ACTION OpenSeperator_action:
ST03_557_Y70_1.MoveInit:=TRUE;		(* Zuführung Vereinzler AST/GST *)
END_ACTION

ACTION Kamera_nicht_bb_entry:
MessageHandler.ClearMessageLines(sVisu:=Visu.Message);
END_ACTION

ACTION Kamera_nicht_bb_action:
MessageHandler.Msg.ID:='PM152';
MessageHandler.Msg.Name:='Check Camera';
MessageHandler.Msg.Text:='Sesopart Kamera ist nicht betriebsbereit';
MessageHandler.Msg.Color:=Color.red;
MessageHandler.Msg.Station:=1;


MessageHandler(
	Prio:=2, 							(*1=highest, .. , 4=lowest*)
	Btn1Addr:=ADR(MsgOk),			(*Address of Button1 , if Zero then Button is unvisible*)
	Btn2Addr:=,						(*Address of Button2 , if Zero then Button is unvisible*)
	sVisu:=Visu.Message);
END_ACTION

ACTION Kamera_nicht_bb_exit:
MsgOk:=FALSE;
MsgCancel:=FALSE;
ST02_DT_95_A1.b_quitt:=TRUE;
END_ACTION

ACTION Wait_for_Part_entry:
ProcessMessage01:='';
Delay.IN:=FALSE;
Delay();
END_ACTION

ACTION Wait_for_Part_action:
ProcessMessage01:='1IM9';(*warte auf Teil in Stopper*)
Delay.IN:=ST03_556_B69_6.BitInToCheck; 		(*  ISK an Stopper.*)
Delay.PT:=T#500ms;
Delay();
END_ACTION

ACTION Wait_for_Part_exit:
ProcessMessage01:='';
END_ACTION

ACTION Close_Seperator_action:
ST03_557_Y70_1.MoveWork:=TRUE;		(*Zuführung Vereinzler AST/GST *)
END_ACTION

ACTION Open_Stopper_action:
ST03_557_Y70_2.MoveWork:=TRUE;		(* Züführung Stopper AST/GST *)
END_ACTION

ACTION Wait_for_Part__entry:
ProcessMessage01:='';
Delay(IN:=FALSE);
END_ACTION

ACTION Wait_for_Part__action:
ProcessMessage01:='1IM10';(*warte auf Teil in Abholposition*)
Delay(	IN:=	ST03_Init_AbholPos.RoboPos31,
		PT:=T#500ms);
END_ACTION

ACTION Wait_for_Part__exit:
ProcessMessage01:='';
Delay(IN:=FALSE);
END_ACTION

ACTION Close_Stopper_action:
ST03_557_Y70_2.MoveInit:=TRUE;		(* Züführung Stopper AST/GST *)
END_ACTION

ACTION Open_Seperator_action:
ST03_557_Y70_1.MoveInit:=TRUE;		(* Zuführung Vereinzler AST/GST *)
END_ACTION

ACTION Robot01_Pos31_action:
Robot01.PosNo:=POS_WT_POS1;
Robot01.PosOffset:=gRobotOffset;
Robot01.Override:=MP.ST00.Override;
Robot01.SetToolOn:=FALSE;
Robot01.SetToolOff:=TRUE;
Robot01.ExecuteMove:=TRUE;
END_ACTION

ACTION Robot01_Pos31_exit:
gRob01GripState:=PART_CAM;
FOR i:=1 TO NO_OF_RESULT BY 1 DO
	Result[i]:=0;
END_FOR
END_ACTION

ACTION Robot01_Pos41_entry:
RepeatCounter:=0;
END_ACTION

ACTION Robot01_Pos41_action:
Robot01.PosNo:=POS_CAM_POS1;
Robot01.PosOffset:=gRobotOffset;
Robot01.Override:=MP.ST00.Override;
Robot01.SetToolOn:=FALSE;
Robot01.SetToolOff:=TRUE;
Robot01.ExecuteMove:=TRUE;
Pos:=1;
END_ACTION

ACTION Robot01_Pos45_entry:
RepeatCounter:=0;
END_ACTION

ACTION Robot01_Pos45_action:
Robot01.PosNo:=POS_CAM_POS2;
Robot01.PosOffset:=gRobotOffset;
Robot01.Override:=MP.ST00.Override;
Robot01.SetToolOn:=FALSE;
Robot01.SetToolOff:=TRUE;
Robot01.ExecuteMove:=TRUE;
Pos:=2;
END_ACTION

ACTION Start_Sensopart_action:
ST03_8_100_A1.JobNo := TD.Sensopart_CamProgNo ;
ST03_8_100_A1.st_ctrl_in.b_start := TRUE;
END_ACTION

ACTION WaitDone_entry:
ST03_8_100_A1.st_ctrl_in.b_start := FALSE;
RepeatCounter:=RepeatCounter+1;
END_ACTION

ACTION ResultCam_entry:
IF 	(ST03_8_100_A1.b_Kam_Pruef_IO AND	 (*Kamera Farberkennung*)
	NOT ST03_8_100_A1.b_Kam_Pruef_NIO) THEN
	Result[Pos]:=RESULT_OK;
ELSE
	Result[Pos]:=RESULT_NOK;
END_IF
END_ACTION

ACTION Result2_entry:
FOR i:=1 TO NO_OF_RESULT BY 1 DO
	Result[i]:=RESULT_OK;
END_FOR
END_ACTION

ACTION Result_Counter_entry:
FOR i:=100 TO 2 BY-1 DO
   	NokPercent[i] := NokPercent[i-1];
END_FOR

ResultOk:=TRUE;
FOR i:=1 TO NO_OF_RESULT BY 1 DO
	IF	ResultOk AND Result[i] = RESULT_NOK 	THEN
		ResultOk:=FALSE;
	END_IF
END_FOR

IF 	ResultOk OR
	CamAlwaysOK THEN		(*schreibt immer NOK nur zum Testen*)
	NokCounter:=0;
	NokPercent[1] := FALSE;
	gRob01GripState:=PART_OK;
ELSE
	NokCounter:=NokCounter+1;
	NokPercent[1] := TRUE;
	gRob01GripState:=PART_NOK;
END_IF
END_ACTION

ACTION Msg_Cam_entry:
MessageHandler.ClearMessageLines(sVisu:=Visu.Message);
END_ACTION

ACTION Msg_Cam_action:
MessageHandler.Msg.ID:='PM112';
MessageHandler.Msg.Name:='Sensopart Kam.-Erg. Prüfung  n.i.o:';
MessageHandler.Msg.Text:='Sensopart Kam.-Erg. Prüfung  n.i.o: Fehler in Folge';
MessageHandler.Msg.Color:=Color.red;
MessageHandler.Msg.Station:=3;
MessageHandler.MsgButton1Text:='continue';

MessageHandler(
	Prio:=2, 								(*1=highest, .. , 4=lowest*)
	Btn1Addr:=ADR(MsgOk),				(*Address of Button1 , if Zero then Button is unvisible*)
	Btn2Addr:=0(*ADR(MsgCancel)*),			(*Address of Button2 , if Zero then Button is unvisible*)
	sVisu:=Visu.Message);
END_ACTION

ACTION Msg_Cam_exit:
MsgOk:=FALSE;
MsgCancel:=FALSE;
END_ACTION

ACTION CounterReset_entry:
NokCounter:=0;
END_ACTION

ACTION Msg_Cam_Percent_entry:
MessageHandler.ClearMessageLines(sVisu:=Visu.Message);
END_ACTION

ACTION Msg_Cam_Percent_action:
MessageHandler.Msg.ID:='PM113';
MessageHandler.Msg.Name:='Sensopart Kam.-Erg. Prüfung  n.i.o:';
MessageHandler.Msg.Text:='Sensopart Kam.-Erg. Prüfung  n.i.o:% Fehler';
MessageHandler.Msg.Color:=Color.red;
MessageHandler.Msg.Station:=3;
MessageHandler.MsgButton1Text:='continue';

MessageHandler(
	Prio:=2, 								(*1=highest, .. , 4=lowest*)
	Btn1Addr:=ADR(MsgOk),				(*Address of Button1 , if Zero then Button is unvisible*)
	Btn2Addr:=0(*ADR(MsgCancel)*),			(*Address of Button2 , if Zero then Button is unvisible*)
	sVisu:=Visu.Message);
END_ACTION

ACTION Msg_Cam_Percent_exit:
MsgOk:=FALSE;
MsgCancel:=FALSE;
END_ACTION

ACTION CounterResetP_entry:
NokCounter:=0;
(*Percent Register löschen*)
FOR i:=1 TO 100 BY 1 DO
  NokPercent[i]:= FALSE;
END_FOR
END_ACTION

ACTION Robot01_Park_action:
Robot01.PosNo:=POS_PARK;
Robot01.PosOffset:=gRobotOffset;
Robot01.Override:=MP.ST00.Override;
Robot01.SetToolOn:=FALSE;
Robot01.SetToolOff:=TRUE;
Robot01.ExecuteMove:=TRUE;
END_ACTION

ACTION SeqEnd_action:
SFCTime:=TIME_TO_DINT(TIME()-SFCTimeStart);
State:=STATE_WAIT;
END_ACTION

TRANSITION Kamera_betriebsbereit:
(*Kamera Farberkennung*)
(
NOT ST03_8_100_A1.sm_kamera_nicht_bb OR
NOT ST03_8_100_A1.Activated	)
END_TRANSITION

TRANSITION NotPartCam:
gRob01GripState<>PART_CAM
END_TRANSITION

TRANSITION Abholpos leer:
NOT ST03_Init_AbholPos.RoboPos31
END_TRANSITION

TRANSITION PartCam:
TRUE
END_TRANSITION

TRANSITION State Ok:
ST03_557_Y70_2.State=STATE_OK AND	(*Züführung Stopper AST/GST *)
ST03_557_Y70_1.State=STATE_OK			(* Zuführung Vereinzler AST/GST *)
END_TRANSITION

TRANSITION Part Ready:
Delay.Q AND
NOT ST03_Init_AbholPos.RoboPos31 AND
ST03_556_B69_6.BitInToCheck	AND			(*ISK anwesend am Stoper*)
Robot01.ActualArea <> 4
END_TRANSITION

TRANSITION StateOk:
ST03_557_Y70_1.State=STATE_OK AND	(* Zuführung Vereinzler AST/GST *)
Robot01.ActualArea <> 3 AND
Robot01.ActualArea <> 4
END_TRANSITION

TRANSITION State Ok:
ST03_557_Y70_2.State=STATE_OK 	(* Züführung Stopper AST/GST *)
END_TRANSITION

TRANSITION Part Ready:
Delay.Q AND
Robot01.ActualArea <> 4
END_TRANSITION

TRANSITION State Ok:
ST03_557_Y70_2.State=STATE_OK AND	(*Züführung Stopper AST/GST *)
ST03_557_Y70_1.State=STATE_OK			(* Zuführung Vereinzler AST/GST *)
END_TRANSITION

TRANSITION AbholPos:
ST03_556_B69_7. BitInToCheck (*ISK anwesend an Abholposition*)
END_TRANSITION

TRANSITION GripperEmpty:
gRob01GripState=PART_NO AND
Robot01.RemInToolWorkSensor
END_TRANSITION

TRANSITION #StateOK:
Robot01.State=STATE_WAIT AND
gRob01GripState=PART_NO
END_TRANSITION

TRANSITION #StateOK:
Robot01.State=STATE_OK AND
gTipImp
END_TRANSITION

TRANSITION CamActive:
ST03_8_100_A1.Activated
END_TRANSITION

TRANSITION #StateOK:
Robot01.State=STATE_OK AND
gTipImp
END_TRANSITION

TRANSITION #StateOK:
Robot01.State=STATE_OK AND
gTipImp
END_TRANSITION

TRANSITION Busy:
ST03_8_100_A1.st_ctrl_out.b_busy (*Kamera Farberkennung Ehternet*)
END_TRANSITION

TRANSITION Done:
ST03_8_100_A1.st_ctrl_out.b_fertig
END_TRANSITION

TRANSITION io:
Result[Pos]=RESULT_OK
END_TRANSITION

TRANSITION nio:
RepeatCounter>=2
END_TRANSITION

TRANSITION Repeat_:
TRUE
END_TRANSITION

TRANSITION CounterOK:
(NokCounter<MP.ST03.CamNoOfErrors AND
NokCounterPercent < MP.ST02.CamNoOfErrorsPercent) OR
CamAlwaysOk
END_TRANSITION

TRANSITION Nok_Cont:
NokCounter >= MP.ST03.CamNoOfErrors
END_TRANSITION

TRANSITION Nok_Percent:
NokCounterPercent >= MP.ST03.CamNoOfErrorsPercent
END_TRANSITION

TRANSITION PartOK:
gRob01GripState=PART_OK
END_TRANSITION

TRANSITION #StateOK:
Robot01.State=STATE_OK AND
gTipImp
END_TRANSITION

TRANSITION PartNOK:
(*NIO Pos wird im ST03_Main angefahren*)
gRob01GripState=PART_NOK
END_TRANSITION
END_PROGRAM

(* POU Stations/ST_03_Ruestsaetze/ST_03_SFCs/Zufuehrungen/ST03_102pol_neu_Zufuehrung, SFC *)
PROGRAM ST03_102pol_neu_Zufuehrung
VAR_INPUT
	Start					:BOOL;
END_VAR
VAR_OUTPUT
	SFCCurrentPOU			: STRING:='ST03_102pol_neu_Zufuehrung';
	SFCCurrentStep			: STRING:='';
	FB_CurrentStepHistorie	: FB_CurrentStepHistorie;
	SFCTime				: DINT;
	State   					: StateObject	:= STATE_WAIT;
	ResultCam				: ARRAY [1..NO_OF_RESULT] OF StateResult;
	ResultOK				: BOOL;
END_VAR
VAR
	MsgOK				: BOOL;
	MsgCancel			: BOOL;
	SFCRun			: BOOL;
	SFCTimeStart		: TIME;
	Delay				: TON;
	(* Userdefinded area *)

	i					: INT:=1;
	Pos					: INT:= 1;
	RepeatCounter		: INT;
	NokCounter			: INT;
	NokCounterPercent	: INT;
  	NokPercent   		: ARRAY[1..100] OF BOOL;
	CamAlwaysOK		: ARRAY[1..2] OF BOOL:=TRUE,TRUE;		(*schreibt immer OK nur zum Testen*)
END_VAR

VAR CONSTANT
	NO_OF_RESULT	: INT :=4;
END_VAR
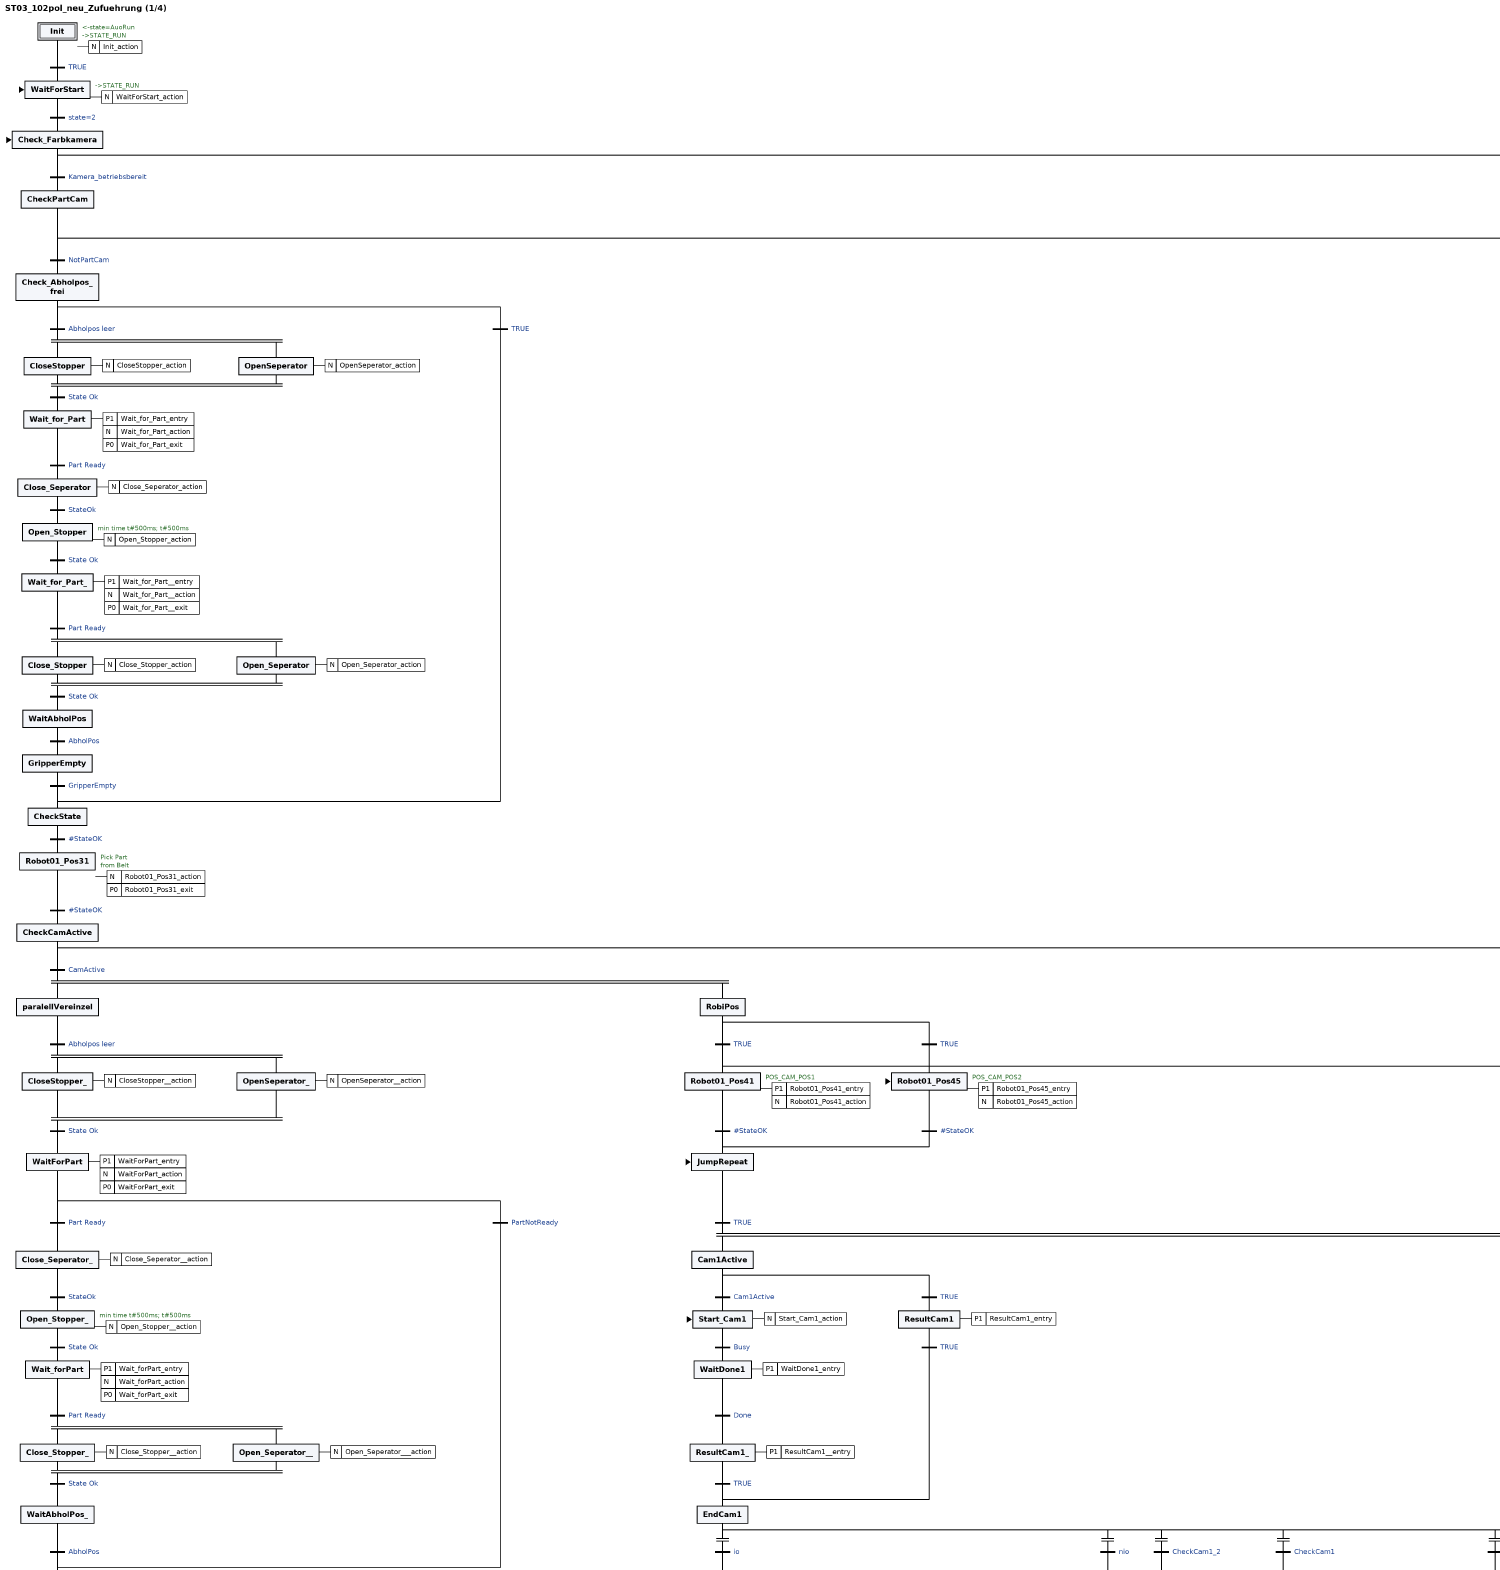
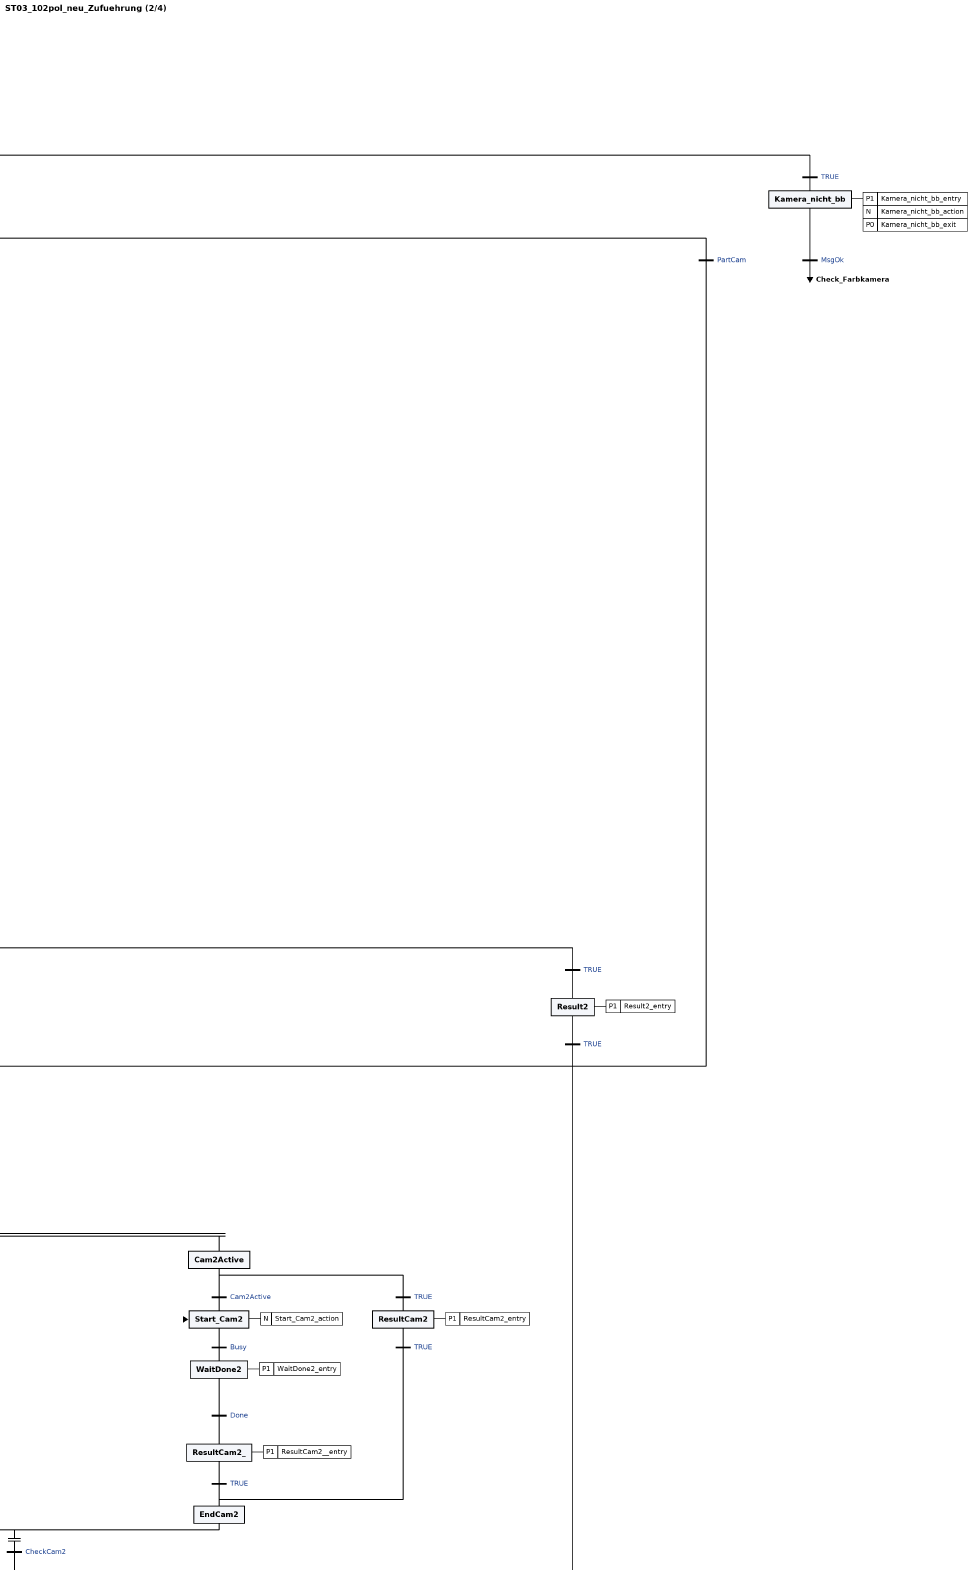
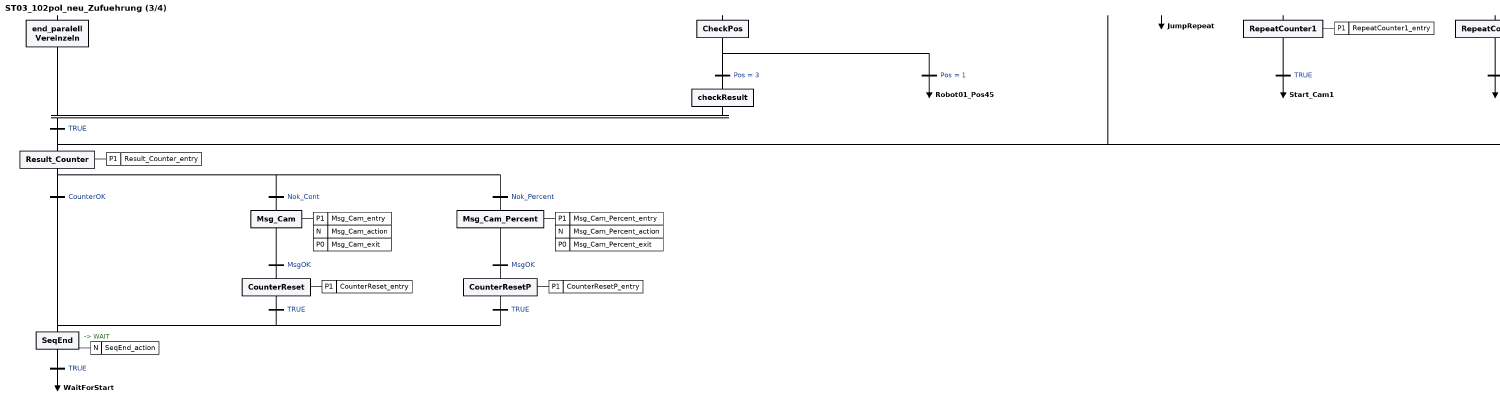
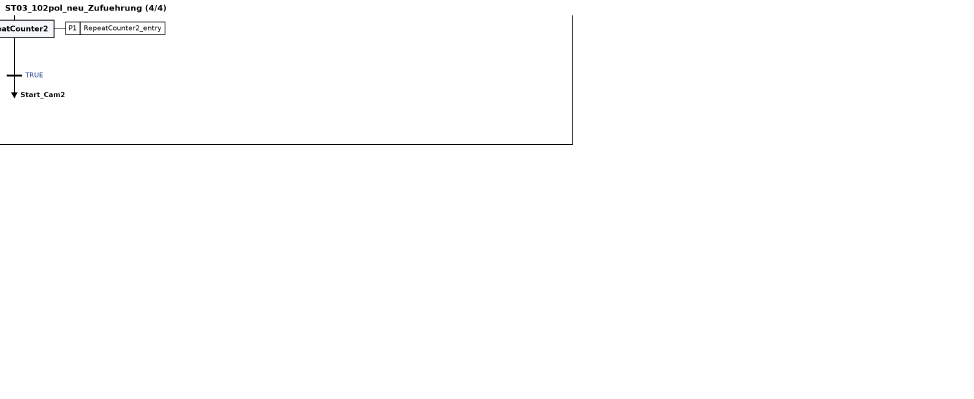
INITIAL_STEP Init: (* <-state=AuoRun / ->STATE_RUN *)
	Init_action(N);
END_STEP
TRANSITION FROM Init TO WaitForStart := TRUE;
END_TRANSITION
STEP WaitForStart: (* ->STATE_RUN *)
	WaitForStart_action(N);
END_STEP
TRANSITION FROM WaitForStart TO Check_Farbkamera := state=2;
END_TRANSITION
STEP Check_Farbkamera:
END_STEP
TRANSITION FROM Check_Farbkamera TO CheckPartCam := Kamera_betriebsbereit;
END_TRANSITION
TRANSITION FROM Check_Farbkamera TO Kamera_nicht_bb := TRUE;
END_TRANSITION
STEP CheckPartCam:
END_STEP
TRANSITION FROM CheckPartCam TO Check_Abholpos_frei := NotPartCam;
END_TRANSITION
TRANSITION FROM CheckPartCam TO Robot01_Pos41 := PartCam;
END_TRANSITION
STEP Check_Abholpos_frei:
END_STEP
TRANSITION FROM Check_Abholpos_frei TO (CloseStopper, OpenSeperator) := Abholpos leer;
END_TRANSITION
TRANSITION FROM Check_Abholpos_frei TO CheckState := TRUE;
END_TRANSITION
STEP CloseStopper:
	CloseStopper_action(N);
END_STEP
STEP OpenSeperator:
	OpenSeperator_action(N);
END_STEP
TRANSITION FROM (CloseStopper, OpenSeperator) TO Wait_for_Part := State Ok;
END_TRANSITION
STEP Kamera_nicht_bb:
	Kamera_nicht_bb_entry(P1);
	Kamera_nicht_bb_action(N);
	Kamera_nicht_bb_exit(P0);
END_STEP
TRANSITION FROM Kamera_nicht_bb TO Check_Farbkamera := MsgOk;
END_TRANSITION
STEP Wait_for_Part:
	Wait_for_Part_entry(P1);
	Wait_for_Part_action(N);
	Wait_for_Part_exit(P0);
END_STEP
TRANSITION FROM Wait_for_Part TO Close_Seperator := Part Ready;
END_TRANSITION
STEP Close_Seperator:
	Close_Seperator_action(N);
END_STEP
TRANSITION FROM Close_Seperator TO Open_Stopper := StateOk;
END_TRANSITION
STEP Open_Stopper: (* min time t#500ms; t#500ms *)
	Open_Stopper_action(N);
END_STEP
TRANSITION FROM Open_Stopper TO Wait_for_Part_ := State Ok;
END_TRANSITION
STEP Wait_for_Part_:
	Wait_for_Part__entry(P1);
	Wait_for_Part__action(N);
	Wait_for_Part__exit(P0);
END_STEP
TRANSITION FROM Wait_for_Part_ TO (Close_Stopper, Open_Seperator) := Part Ready;
END_TRANSITION
STEP Close_Stopper:
	Close_Stopper_action(N);
END_STEP
STEP Open_Seperator:
	Open_Seperator_action(N);
END_STEP
TRANSITION FROM (Close_Stopper, Open_Seperator) TO WaitAbholPos := State Ok;
END_TRANSITION
STEP WaitAbholPos:
END_STEP
TRANSITION FROM WaitAbholPos TO GripperEmpty := AbholPos;
END_TRANSITION
STEP GripperEmpty:
END_STEP
TRANSITION FROM GripperEmpty TO CheckState := GripperEmpty;
END_TRANSITION
STEP CheckState:
END_STEP
TRANSITION FROM CheckState TO Robot01_Pos31 := #StateOK;
END_TRANSITION
STEP Robot01_Pos31: (* Pick Part / from Belt *)
	Robot01_Pos31_action(N);
	Robot01_Pos31_exit(P0);
END_STEP
TRANSITION FROM Robot01_Pos31 TO CheckCamActive := #StateOK;
END_TRANSITION
STEP CheckCamActive:
END_STEP
TRANSITION FROM CheckCamActive TO (paralellVereinzel, RobiPos) := CamActive;
END_TRANSITION
TRANSITION FROM CheckCamActive TO Result2 := TRUE;
END_TRANSITION
STEP paralellVereinzel:
END_STEP
TRANSITION FROM paralellVereinzel TO (CloseStopper_, OpenSeperator_) := Abholpos leer;
END_TRANSITION
STEP CloseStopper_:
	CloseStopper__action(N);
END_STEP
STEP OpenSeperator_:
	OpenSeperator__action(N);
END_STEP
TRANSITION FROM (CloseStopper_, OpenSeperator_) TO WaitForPart := State Ok;
END_TRANSITION
STEP WaitForPart:
	WaitForPart_entry(P1);
	WaitForPart_action(N);
	WaitForPart_exit(P0);
END_STEP
TRANSITION FROM WaitForPart TO Close_Seperator_ := Part Ready;
END_TRANSITION
TRANSITION FROM WaitForPart TO end_paralellVereinzeln := PartNotReady;
END_TRANSITION
STEP Close_Seperator_:
	Close_Seperator__action(N);
END_STEP
TRANSITION FROM Close_Seperator_ TO Open_Stopper_ := StateOk;
END_TRANSITION
STEP Open_Stopper_: (* min time t#500ms; t#500ms *)
	Open_Stopper__action(N);
END_STEP
TRANSITION FROM Open_Stopper_ TO Wait_forPart := State Ok;
END_TRANSITION
STEP Wait_forPart:
	Wait_forPart_entry(P1);
	Wait_forPart_action(N);
	Wait_forPart_exit(P0);
END_STEP
TRANSITION FROM Wait_forPart TO (Close_Stopper_, Open_Seperator__) := Part Ready;
END_TRANSITION
STEP Close_Stopper_:
	Close_Stopper__action(N);
END_STEP
STEP Open_Seperator__:
	Open_Seperator___action(N);
END_STEP
TRANSITION FROM (Close_Stopper_, Open_Seperator__) TO WaitAbholPos_ := State Ok;
END_TRANSITION
STEP WaitAbholPos_:
END_STEP
TRANSITION FROM WaitAbholPos_ TO end_paralellVereinzeln := AbholPos;
END_TRANSITION
STEP end_paralellVereinzeln:
END_STEP
STEP RobiPos:
END_STEP
TRANSITION FROM RobiPos TO Robot01_Pos41 := TRUE;
END_TRANSITION
TRANSITION FROM RobiPos TO Robot01_Pos45 := TRUE;
END_TRANSITION
STEP Robot01_Pos41: (* POS_CAM_POS1 *)
	Robot01_Pos41_entry(P1);
	Robot01_Pos41_action(N);
END_STEP
TRANSITION FROM Robot01_Pos41 TO JumpRepeat := #StateOK;
END_TRANSITION
STEP Robot01_Pos45: (* POS_CAM_POS2 *)
	Robot01_Pos45_entry(P1);
	Robot01_Pos45_action(N);
END_STEP
TRANSITION FROM Robot01_Pos45 TO JumpRepeat := #StateOK;
END_TRANSITION
STEP JumpRepeat:
END_STEP
TRANSITION FROM JumpRepeat TO (Cam1Active, Cam2Active) := TRUE;
END_TRANSITION
STEP Cam1Active:
END_STEP
TRANSITION FROM Cam1Active TO Start_Cam1 := Cam1Active;
END_TRANSITION
TRANSITION FROM Cam1Active TO ResultCam1 := TRUE;
END_TRANSITION
STEP Start_Cam1:
	Start_Cam1_action(N);
END_STEP
TRANSITION FROM Start_Cam1 TO WaitDone1 := Busy;
END_TRANSITION
STEP WaitDone1:
	WaitDone1_entry(P1);
END_STEP
TRANSITION FROM WaitDone1 TO ResultCam1_ := Done;
END_TRANSITION
STEP ResultCam1_:
	ResultCam1__entry(P1);
END_STEP
TRANSITION FROM ResultCam1_ TO EndCam1 := TRUE;
END_TRANSITION
STEP ResultCam1:
	ResultCam1_entry(P1);
END_STEP
TRANSITION FROM ResultCam1 TO EndCam1 := TRUE;
END_TRANSITION
STEP EndCam1:
END_STEP
STEP Cam2Active:
END_STEP
TRANSITION FROM Cam2Active TO Start_Cam2 := Cam2Active;
END_TRANSITION
TRANSITION FROM Cam2Active TO ResultCam2 := TRUE;
END_TRANSITION
STEP Start_Cam2:
	Start_Cam2_action(N);
END_STEP
TRANSITION FROM Start_Cam2 TO WaitDone2 := Busy;
END_TRANSITION
STEP WaitDone2:
	WaitDone2_entry(P1);
END_STEP
TRANSITION FROM WaitDone2 TO ResultCam2_ := Done;
END_TRANSITION
STEP ResultCam2_:
	ResultCam2__entry(P1);
END_STEP
TRANSITION FROM ResultCam2_ TO EndCam2 := TRUE;
END_TRANSITION
STEP ResultCam2:
	ResultCam2_entry(P1);
END_STEP
TRANSITION FROM ResultCam2 TO EndCam2 := TRUE;
END_TRANSITION
STEP EndCam2:
END_STEP
TRANSITION FROM (EndCam1, EndCam2) TO CheckPos := io;
END_TRANSITION
TRANSITION FROM (EndCam1, EndCam2) TO Result_Counter := nio;
END_TRANSITION
TRANSITION FROM (EndCam1, EndCam2) TO JumpRepeat := CheckCam1_2;
END_TRANSITION
TRANSITION FROM (EndCam1, EndCam2) TO RepeatCounter1 := CheckCam1;
END_TRANSITION
TRANSITION FROM (EndCam1, EndCam2) TO RepeatCounter2 := CheckCam2;
END_TRANSITION
STEP RepeatCounter1:
	RepeatCounter1_entry(P1);
END_STEP
TRANSITION FROM RepeatCounter1 TO Start_Cam1 := TRUE;
END_TRANSITION
STEP RepeatCounter2:
	RepeatCounter2_entry(P1);
END_STEP
TRANSITION FROM RepeatCounter2 TO Start_Cam2 := TRUE;
END_TRANSITION
STEP CheckPos:
END_STEP
TRANSITION FROM CheckPos TO checkResult := Pos = 3;
END_TRANSITION
TRANSITION FROM CheckPos TO Robot01_Pos45 := Pos = 1;
END_TRANSITION
STEP checkResult:
END_STEP
TRANSITION FROM (end_paralellVereinzeln, checkResult) TO Result_Counter := TRUE;
END_TRANSITION
STEP Result2:
	Result2_entry(P1);
END_STEP
TRANSITION FROM Result2 TO Result_Counter := TRUE;
END_TRANSITION
STEP Result_Counter:
	Result_Counter_entry(P1);
END_STEP
TRANSITION FROM Result_Counter TO SeqEnd := CounterOK;
END_TRANSITION
TRANSITION FROM Result_Counter TO Msg_Cam := Nok_Cont;
END_TRANSITION
TRANSITION FROM Result_Counter TO Msg_Cam_Percent := Nok_Percent;
END_TRANSITION
STEP Msg_Cam:
	Msg_Cam_entry(P1);
	Msg_Cam_action(N);
	Msg_Cam_exit(P0);
END_STEP
TRANSITION FROM Msg_Cam TO CounterReset := MsgOK;
END_TRANSITION
STEP CounterReset:
	CounterReset_entry(P1);
END_STEP
TRANSITION FROM CounterReset TO SeqEnd := TRUE;
END_TRANSITION
STEP Msg_Cam_Percent:
	Msg_Cam_Percent_entry(P1);
	Msg_Cam_Percent_action(N);
	Msg_Cam_Percent_exit(P0);
END_STEP
TRANSITION FROM Msg_Cam_Percent TO CounterResetP := MsgOK;
END_TRANSITION
STEP CounterResetP:
	CounterResetP_entry(P1);
END_STEP
TRANSITION FROM CounterResetP TO SeqEnd := TRUE;
END_TRANSITION
STEP SeqEnd: (* -> WAIT *)
	SeqEnd_action(N);
END_STEP
TRANSITION FROM SeqEnd TO WaitForStart := TRUE;
END_TRANSITION

ACTION Init_action:
Start:=FALSE;
State:=STATE_WAIT;
MsgOK:=FALSE;
MsgCancel:=FALSE;
SFCRun:=FALSE;
NokCounter:=0;
i:=1;
Pos:=1;
FOR i:=1 TO NO_OF_RESULT BY 1 DO
	ResultCam[i]:=RESULT_NON;
END_FOR
END_ACTION

ACTION WaitForStart_action:
IF 	Start   THEN
	State:=STATE_RUN;
	SFCTimeStart:=TIME();
	Start:=FALSE;
	FOR i:=1 TO NO_OF_RESULT BY 1 DO
		ResultCam[i]:=RESULT_NON;
	END_FOR
	i:=1;
	Pos:=1;
ELSE
	State:=STATE_WAIT;
	MsgOK:=FALSE;
	MsgCancel:=FALSE;
	SFCRun:=FALSE;
END_IF
END_ACTION

ACTION CloseStopper_action:
ST03_557_Y70_2.MoveInit:=TRUE;		(* Züführung Stopper AST/GST *)
END_ACTION

ACTION OpenSeperator_action:
ST03_557_Y70_1.MoveInit:=TRUE;		(* Zuführung Vereinzler AST/GST *)
END_ACTION

ACTION Kamera_nicht_bb_entry:
MessageHandler.ClearMessageLines(sVisu:=Visu.Message);
END_ACTION

ACTION Kamera_nicht_bb_action:
MessageHandler.Msg.ID:='PM152';
MessageHandler.Msg.Name:='Check Camera';
MessageHandler.Msg.Text:='Sesopart Kamera ist nicht betriebsbereit';
MessageHandler.Msg.Color:=Color.red;
MessageHandler.Msg.Station:=1;


MessageHandler(
	Prio:=2, 							(*1=highest, .. , 4=lowest*)
	Btn1Addr:=ADR(MsgOk),			(*Address of Button1 , if Zero then Button is unvisible*)
	Btn2Addr:=,						(*Address of Button2 , if Zero then Button is unvisible*)
	sVisu:=Visu.Message);
END_ACTION

ACTION Kamera_nicht_bb_exit:
MsgOk:=FALSE;
MsgCancel:=FALSE;
ST02_DT_95_A1.b_quitt:=TRUE;
END_ACTION

ACTION Wait_for_Part_entry:
ProcessMessage01:='';
Delay.IN:=FALSE;
Delay();
END_ACTION

ACTION Wait_for_Part_action:
ProcessMessage01:='1IM9';(*warte auf Teil in Stopper*)
Delay.IN:=ST03_556_B69_6.BitInToCheck; 		(*  ISK an Stopper.*)
Delay.PT:=T#500ms;
Delay();
END_ACTION

ACTION Wait_for_Part_exit:
ProcessMessage01:='';
END_ACTION

ACTION Close_Seperator_action:
ST03_557_Y70_1.MoveWork:=TRUE;		(*Zuführung Vereinzler AST/GST *)
END_ACTION

ACTION Open_Stopper_action:
ST03_557_Y70_2.MoveWork:=TRUE;		(* Züführung Stopper AST/GST *)
END_ACTION

ACTION Wait_for_Part__entry:
ProcessMessage01:='';
Delay(IN:=FALSE);
END_ACTION

ACTION Wait_for_Part__action:
ProcessMessage01:='1IM10';(*warte auf Teil in Abholposition*)
Delay(	IN:=	ST03_Init_AbholPos.RoboPos31,
		PT:=T#500ms);
END_ACTION

ACTION Wait_for_Part__exit:
ProcessMessage01:='';
Delay(IN:=FALSE);
END_ACTION

ACTION Close_Stopper_action:
ST03_557_Y70_2.MoveInit:=TRUE;		(* Züführung Stopper AST/GST *)
END_ACTION

ACTION Open_Seperator_action:
ST03_557_Y70_1.MoveInit:=TRUE;		(* Zuführung Vereinzler AST/GST *)
END_ACTION

ACTION Robot01_Pos31_action:
Robot01.PosNo:=POS_WT_POS1;
Robot01.PosOffset:=gRobotOffset;
Robot01.Override:=MP.ST00.Override;
Robot01.SetToolOn:=FALSE;
Robot01.SetToolOff:=TRUE;
Robot01.ExecuteMove:=TRUE;
END_ACTION

ACTION Robot01_Pos31_exit:
gRob01GripState:=PART_CAM;

FOR i:=1 TO NO_OF_RESULT BY 1 DO
	ResultCam[i]:=0;
END_FOR
END_ACTION

ACTION CloseStopper__action:
ST03_557_Y70_2.MoveInit:=TRUE;		(* Züführung Stopper AST/GST *)
END_ACTION

ACTION OpenSeperator__action:
ST03_557_Y70_1.MoveInit:=TRUE;		(* Zuführung Vereinzler AST/GST *)
END_ACTION

ACTION WaitForPart_entry:
ProcessMessage01:='';
Delay();
END_ACTION

ACTION WaitForPart_action:
ProcessMessage01:='1IM9';(*warte auf Teil in Stopper*)
Delay();
END_ACTION

ACTION WaitForPart_exit:
ProcessMessage01:='';
END_ACTION

ACTION Close_Seperator__action:
ST03_557_Y70_1.MoveWork:=TRUE;		(*Zuführung Vereinzler AST/GST *)
END_ACTION

ACTION Open_Stopper__action:
ST03_557_Y70_2.MoveWork:=TRUE;		(* Züführung Stopper AST/GST *)
END_ACTION

ACTION Wait_forPart_entry:
ProcessMessage01:='';
Delay(IN:=FALSE);
END_ACTION

ACTION Wait_forPart_action:
ProcessMessage01:='1IM10';(*warte auf Teil in Abholposition*)
Delay(	IN:=	ST03_Init_AbholPos.RoboPos31,
		PT:=T#500ms);
END_ACTION

ACTION Wait_forPart_exit:
ProcessMessage01:='';
Delay(IN:=FALSE);
END_ACTION

ACTION Close_Stopper__action:
ST03_557_Y70_2.MoveInit:=TRUE;		(* Züführung Stopper AST/GST *)
END_ACTION

ACTION Open_Seperator___action:
ST03_557_Y70_1.MoveInit:=TRUE;		(* Zuführung Vereinzler AST/GST *)
END_ACTION

ACTION Robot01_Pos41_entry:
RepeatCounter:=1;
END_ACTION

ACTION Robot01_Pos41_action:
Robot01.PosNo:=POS_CAM_POS1;
Robot01.PosOffset:=gRobotOffset;
Robot01.Override:=MP.ST00.Override;
Robot01.SetToolOn:=FALSE;
Robot01.SetToolOff:=TRUE;
Robot01.ExecuteMove:=TRUE;
Pos:=1;
END_ACTION

ACTION Robot01_Pos45_entry:
RepeatCounter:=0;
END_ACTION

ACTION Robot01_Pos45_action:
Robot01.PosNo:=POS_CAM_POS2;
Robot01.PosOffset:=gRobotOffset;
Robot01.Override:=MP.ST00.Override;
Robot01.SetToolOn:=FALSE;
Robot01.SetToolOff:=TRUE;
Robot01.ExecuteMove:=TRUE;
Pos:=3;
END_ACTION

ACTION Start_Cam1_action:
IF 	Pos =1 THEN
	ST03_8_100_A1.JobNo := TD.Sensopart_CamProgNo ;
ELSIF
	Pos = 3 THEN
	ST03_8_100_A1.JobNo := TD.Sensopart_CamProgNo + 1 ;
END_IF
ST03_8_100_A1.st_ctrl_in.b_start := TRUE;
END_ACTION

ACTION WaitDone1_entry:
ST03_8_100_A1.st_ctrl_in.b_start := FALSE;
RepeatCounter:=RepeatCounter+1;
END_ACTION

ACTION ResultCam1__entry:
IF 	(ST03_8_100_A1.b_Kam_Pruef_IO AND	 (*Kamera Farberkennung*)
	NOT ST03_8_100_A1.b_Kam_Pruef_NIO) OR
	CamAlwaysOK[1] THEN
	ResultCam[Pos]:=RESULT_OK;
ELSE
	ResultCam[Pos]:=RESULT_NOK;
END_IF
END_ACTION

ACTION ResultCam1_entry:
ResultCam[Pos]:=RESULT_OK;
END_ACTION

ACTION Start_Cam2_action:
IF 	Pos =1 THEN
	ST03_8_103_A1.JobNo := TD.Sensopart2_CamProgNo ;
ELSIF
	Pos = 3 THEN
	ST03_8_103_A1.JobNo := TD.Sensopart2_CamProgNo + 1 ;
END_IF
ST03_8_103_A1.st_ctrl_in.b_start := TRUE;
END_ACTION

ACTION WaitDone2_entry:
ST03_8_103_A1.st_ctrl_in.b_start := FALSE;
END_ACTION

ACTION ResultCam2__entry:
IF 	(ST03_8_103_A1.b_Kam_Pruef_IO AND	 (*Kamera Flügel*)
	NOT ST03_8_103_A1.b_Kam_Pruef_NIO) OR
	CamAlwaysOK[2] THEN
	ResultCam[Pos+1]:=RESULT_OK;
ELSE
	ResultCam[Pos+1]:=RESULT_NOK;
END_IF
END_ACTION

ACTION ResultCam2_entry:
ResultCam[Pos+1]:=RESULT_OK;
END_ACTION

ACTION RepeatCounter1_entry:
RepeatCounter:=RepeatCounter+1;
END_ACTION

ACTION RepeatCounter2_entry:
RepeatCounter:=RepeatCounter+1;
END_ACTION

ACTION Result2_entry:
FOR i:=1 TO NO_OF_RESULT BY 1 DO
	ResultCam[i]:=RESULT_OK;
END_FOR
END_ACTION

ACTION Result_Counter_entry:
FOR i:=100 TO 2 BY-1 DO
   	NokPercent[i] := NokPercent[i-1];
END_FOR

ResultOk:=TRUE;
FOR i:=1 TO NO_OF_RESULT BY 1 DO
	IF	ResultOk AND ResultCam[i] = RESULT_NOK 	THEN
		ResultOk:=FALSE;
	END_IF
END_FOR


IF 	ResultOk  THEN
	NokCounter:=0;
	NokPercent[1] := FALSE;
	gRob01GripState:=PART_OK;
ELSE
	NokCounter:=NokCounter+1;
	NokPercent[1] := TRUE;
	gRob01GripState:=PART_NOK;
END_IF
END_ACTION

ACTION Msg_Cam_entry:
MessageHandler.ClearMessageLines(sVisu:=Visu.Message);
END_ACTION

ACTION Msg_Cam_action:
MessageHandler.Msg.ID:='PM112';
MessageHandler.Msg.Name:='Sensopart Kam.-Erg. Prüfung  n.i.o:';
MessageHandler.Msg.Text:='Sensopart Kam.-Erg. Prüfung  n.i.o: Fehler in Folge';
MessageHandler.Msg.Color:=Color.red;
MessageHandler.Msg.Station:=3;
MessageHandler.MsgButton1Text:='continue';

MessageHandler(
	Prio:=2, 								(*1=highest, .. , 4=lowest*)
	Btn1Addr:=ADR(MsgOk),				(*Address of Button1 , if Zero then Button is unvisible*)
	Btn2Addr:=0(*ADR(MsgCancel)*),			(*Address of Button2 , if Zero then Button is unvisible*)
	sVisu:=Visu.Message);
END_ACTION

ACTION Msg_Cam_exit:
MsgOk:=FALSE;
MsgCancel:=FALSE;
END_ACTION

ACTION CounterReset_entry:
NokCounter:=0;
END_ACTION

ACTION Msg_Cam_Percent_entry:
MessageHandler.ClearMessageLines(sVisu:=Visu.Message);
END_ACTION

ACTION Msg_Cam_Percent_action:
MessageHandler.Msg.ID:='PM113';
MessageHandler.Msg.Name:='Sensopart Kam.-Erg. Prüfung  n.i.o:';
MessageHandler.Msg.Text:='Sensopart Kam.-Erg. Prüfung  n.i.o:% Fehler';
MessageHandler.Msg.Color:=Color.red;
MessageHandler.Msg.Station:=3;
MessageHandler.MsgButton1Text:='continue';

MessageHandler(
	Prio:=2, 								(*1=highest, .. , 4=lowest*)
	Btn1Addr:=ADR(MsgOk),				(*Address of Button1 , if Zero then Button is unvisible*)
	Btn2Addr:=0(*ADR(MsgCancel)*),			(*Address of Button2 , if Zero then Button is unvisible*)
	sVisu:=Visu.Message);
END_ACTION

ACTION Msg_Cam_Percent_exit:
MsgOk:=FALSE;
MsgCancel:=FALSE;
END_ACTION

ACTION CounterResetP_entry:
NokCounter:=0;
(*Percent Register löschen*)
FOR i:=1 TO 100 BY 1 DO
  NokPercent[i]:= FALSE;
END_FOR
END_ACTION

ACTION SeqEnd_action:
SFCTime:=TIME_TO_DINT(TIME()-SFCTimeStart);
State:=STATE_WAIT;
END_ACTION

TRANSITION Kamera_betriebsbereit:
(*Kamera Farberkennung*)
(
NOT ST03_8_100_A1.sm_kamera_nicht_bb OR
NOT ST03_8_100_A1.Activated	) AND
(
NOT ST03_8_103_A1.sm_kamera_nicht_bb OR
NOT ST03_8_103_A1.Activated	)
END_TRANSITION

TRANSITION NotPartCam:
gRob01GripState<>PART_CAM
END_TRANSITION

TRANSITION Abholpos leer:
NOT ST03_Init_AbholPos.RoboPos31
END_TRANSITION

TRANSITION PartCam:
TRUE
END_TRANSITION

TRANSITION State Ok:
ST03_557_Y70_2.State=STATE_OK AND	(*Züführung Stopper AST/GST *)
ST03_557_Y70_1.State=STATE_OK			(* Zuführung Vereinzler AST/GST *)
END_TRANSITION

TRANSITION Part Ready:
Delay.Q AND
NOT ST03_Init_AbholPos.RoboPos31 AND
ST03_556_B69_6.BitInToCheck	AND			(*ISK anwesend am Stoper*)
Robot01.ActualArea <> 4
END_TRANSITION

TRANSITION StateOk:
ST03_557_Y70_1.State=STATE_OK AND	(* Zuführung Vereinzler AST/GST *)
Robot01.ActualArea <> 4
END_TRANSITION

TRANSITION State Ok:
ST03_557_Y70_2.State=STATE_OK 	(* Züführung Stopper AST/GST *)
END_TRANSITION

TRANSITION Part Ready:
Delay.Q AND
Robot01.ActualArea <> 4
END_TRANSITION

TRANSITION State Ok:
ST03_557_Y70_2.State=STATE_OK AND	(*Züführung Stopper AST/GST *)
ST03_557_Y70_1.State=STATE_OK			(* Zuführung Vereinzler AST/GST *)
END_TRANSITION

TRANSITION AbholPos:
ST03_Init_AbholPos.RoboPos31 	(*ISK  auf Übergabeposition *)
END_TRANSITION

TRANSITION GripperEmpty:
gRob01GripState=PART_NO AND
Robot01.RemInToolWorkSensor
END_TRANSITION

TRANSITION #StateOK:
Robot01.State=STATE_WAIT AND
gRob01GripState=PART_NO
END_TRANSITION

TRANSITION #StateOK:
Robot01.State=STATE_OK AND
gTipImp
END_TRANSITION

TRANSITION CamActive:
ST03_8_100_A1.Activated OR
ST03_8_103_A1.Activated
END_TRANSITION

TRANSITION Abholpos leer:
NOT ST03_Init_AbholPos.RoboPos31 AND
Robot01.ActualArea <> 4
END_TRANSITION

TRANSITION State Ok:
ST03_557_Y70_2.State=STATE_OK AND	(*Züführung Stopper AST/GST *)
ST03_557_Y70_1.State=STATE_OK			(* Zuführung Vereinzler AST/GST *)
END_TRANSITION

TRANSITION Part Ready:
NOT ST03_Init_AbholPos.RoboPos31 AND
ST03_556_B69_6.BitInToCheck	AND			(*ISK anwesend am Stoper*)
Robot01.ActualArea <> 4
END_TRANSITION

TRANSITION StateOk:
ST03_557_Y70_1.State=STATE_OK AND	(* Zuführung Vereinzler AST/GST *)
Robot01.ActualArea <> 4
END_TRANSITION

TRANSITION State Ok:
ST03_557_Y70_2.State=STATE_OK 	(* Züführung Stopper AST/GST *)
END_TRANSITION

TRANSITION Part Ready:
Delay.Q AND
Robot01.ActualArea <> 4
END_TRANSITION

TRANSITION State Ok:
ST03_557_Y70_2.State=STATE_OK AND	(*Züführung Stopper AST/GST *)
ST03_557_Y70_1.State=STATE_OK			(* Zuführung Vereinzler AST/GST *)
END_TRANSITION

TRANSITION AbholPos:
ST03_Init_AbholPos.RoboPos31 	(*ISK  auf Übergabeposition *)
END_TRANSITION

TRANSITION PartNotReady:
NOT ST03_556_B69_6.BitInToCheck 		(*  ISK an Stopper.*)
END_TRANSITION

TRANSITION #StateOK:
Robot01.State=STATE_OK AND
gTipImp
END_TRANSITION

TRANSITION #StateOK:
Robot01.State=STATE_OK AND
gTipImp
END_TRANSITION

TRANSITION Cam1Active:
ST03_8_100_A1.Activated
END_TRANSITION

TRANSITION Busy:
ST03_8_100_A1.st_ctrl_out.b_busy (*Kamera Farberkennung Ehternet*)
END_TRANSITION

TRANSITION Done:
ST03_8_100_A1.st_ctrl_out.b_fertig
END_TRANSITION

TRANSITION Cam2Active:
ST03_8_103_A1.Activated
END_TRANSITION

TRANSITION Busy:
ST03_8_103_A1.st_ctrl_out.b_busy (*Kamera Farberkennung Ehternet*)
END_TRANSITION

TRANSITION Done:
ST03_8_103_A1.st_ctrl_out.b_fertig
END_TRANSITION

TRANSITION io:
ResultCam[Pos]=RESULT_OK AND
ResultCam[Pos+1]=RESULT_OK
END_TRANSITION

TRANSITION nio:
RepeatCounter>=2
END_TRANSITION

TRANSITION CheckCam1_2:
ResultCam[Pos]=RESULT_NOK AND
ResultCam[Pos+1]=RESULT_NOK
END_TRANSITION

TRANSITION CheckCam1:
ResultCam[Pos]=RESULT_NOK
END_TRANSITION

TRANSITION CheckCam2:
ResultCam[Pos+1]=RESULT_NOK
END_TRANSITION

TRANSITION CounterOK:
NokCounter<MP.ST03.CamNoOfErrors AND
NokCounterPercent < MP.ST02.CamNoOfErrorsPercent
END_TRANSITION

TRANSITION Nok_Cont:
NokCounter >= MP.ST03.CamNoOfErrors
END_TRANSITION

TRANSITION Nok_Percent:
NokCounterPercent >= MP.ST03.CamNoOfErrorsPercent
END_TRANSITION
END_PROGRAM

(* POU Stations/ST_03_Ruestsaetze/ST_03_SFCs/Zufuehrungen/ST03_268_RP_Zufuehrung, SFC *)
 PROGRAM ST03_268_RP_Zufuehrung
VAR_OUTPUT
	SFCCurrentPOU			: STRING:='ST03_268_RP_Zufuehrung';
	SFCCurrentStep			: STRING:='';
	FB_CurrentStepHistorie	:FB_CurrentStepHistorie;
	SFCTime					: DINT;
	State   				: StateObject	:= STATE_WAIT;
	Result  				: StateResult;
END_VAR
VAR_INPUT
	Start					:BOOL;
END_VAR
VAR
	MsgOK				: BOOL;
	MsgCancel			: BOOL;
	SFCRun			: BOOL;
	SFCTimeStart		: TIME;
	Delay				: TON;
	Delay2				: TON;
	(* Userdefinded area *)

END_VAR
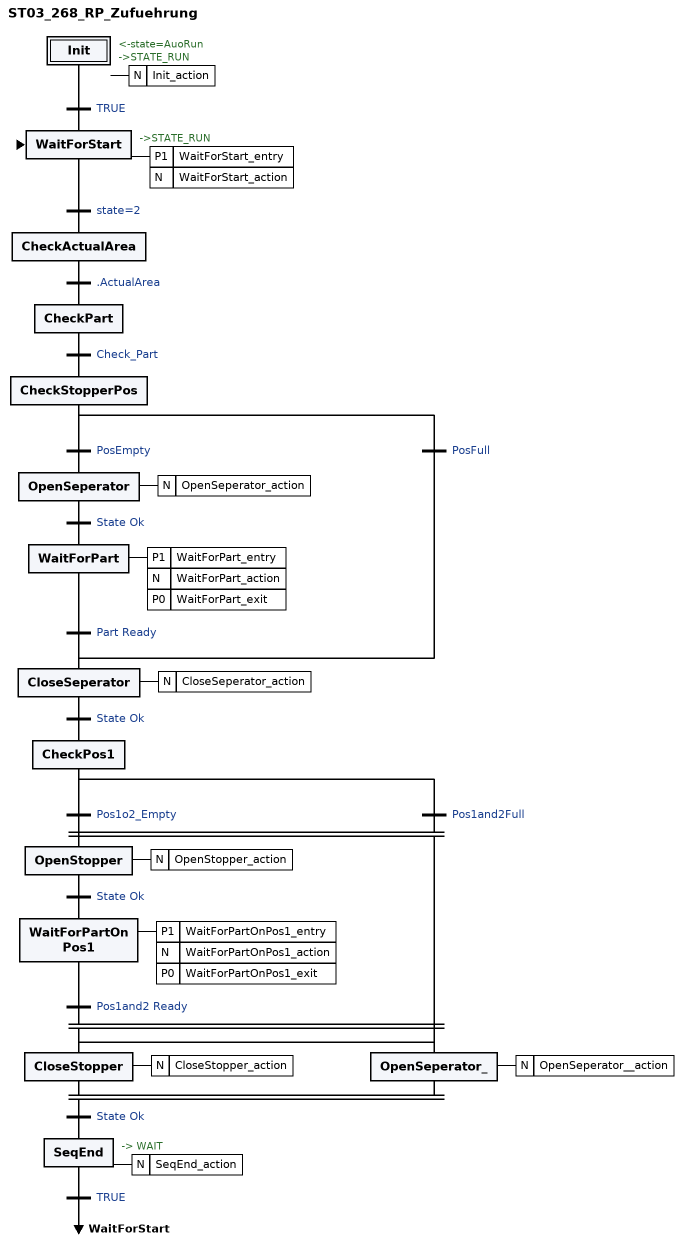
INITIAL_STEP Init: (* <-state=AuoRun / ->STATE_RUN *)
	Init_action(N);
END_STEP
TRANSITION FROM Init TO WaitForStart := TRUE;
END_TRANSITION
STEP WaitForStart: (* ->STATE_RUN *)
	WaitForStart_entry(P1);
	WaitForStart_action(N);
END_STEP
TRANSITION FROM WaitForStart TO CheckActualArea := state=2;
END_TRANSITION
STEP CheckActualArea:
END_STEP
TRANSITION FROM CheckActualArea TO CheckPart := .ActualArea;
END_TRANSITION
STEP CheckPart:
END_STEP
TRANSITION FROM CheckPart TO CheckStopperPos := Check_Part;
END_TRANSITION
STEP CheckStopperPos:
END_STEP
TRANSITION FROM CheckStopperPos TO OpenSeperator := PosEmpty;
END_TRANSITION
TRANSITION FROM CheckStopperPos TO CloseSeperator := PosFull;
END_TRANSITION
STEP OpenSeperator:
	OpenSeperator_action(N);
END_STEP
TRANSITION FROM OpenSeperator TO WaitForPart := State Ok;
END_TRANSITION
STEP WaitForPart:
	WaitForPart_entry(P1);
	WaitForPart_action(N);
	WaitForPart_exit(P0);
END_STEP
TRANSITION FROM WaitForPart TO CloseSeperator := Part Ready;
END_TRANSITION
STEP CloseSeperator:
	CloseSeperator_action(N);
END_STEP
TRANSITION FROM CloseSeperator TO CheckPos1 := State Ok;
END_TRANSITION
STEP CheckPos1:
END_STEP
TRANSITION FROM CheckPos1 TO OpenStopper := Pos1o2_Empty;
END_TRANSITION
TRANSITION FROM CheckPos1 TO (CloseStopper, OpenSeperator_) := Pos1and2Full;
END_TRANSITION
STEP OpenStopper:
	OpenStopper_action(N);
END_STEP
TRANSITION FROM OpenStopper TO WaitForPartOnPos1 := State Ok;
END_TRANSITION
STEP WaitForPartOnPos1:
	WaitForPartOnPos1_entry(P1);
	WaitForPartOnPos1_action(N);
	WaitForPartOnPos1_exit(P0);
END_STEP
TRANSITION FROM WaitForPartOnPos1 TO (CloseStopper, OpenSeperator_) := Pos1and2 Ready;
END_TRANSITION
STEP CloseStopper:
	CloseStopper_action(N);
END_STEP
STEP OpenSeperator_:
	OpenSeperator__action(N);
END_STEP
TRANSITION FROM (CloseStopper, OpenSeperator_) TO SeqEnd := State Ok;
END_TRANSITION
STEP SeqEnd: (* -> WAIT *)
	SeqEnd_action(N);
END_STEP
TRANSITION FROM SeqEnd TO WaitForStart := TRUE;
END_TRANSITION

ACTION Init_action:
Start:=FALSE;
State:=STATE_WAIT;
MsgOK:=FALSE;
MsgCancel:=FALSE;
SFCRun:=FALSE;
Result:=RESULT_NON;
END_ACTION

ACTION WaitForStart_entry:
;
END_ACTION

ACTION WaitForStart_action:
IF 	Start   THEN
	State:=STATE_RUN;
	Result:=RESULT_NON;
	SFCTimeStart:=TIME();
	Start:=FALSE;
ELSE
	State:=STATE_WAIT;
	MsgOK:=FALSE;
	MsgCancel:=FALSE;
	SFCRun:=FALSE;
END_IF
END_ACTION

ACTION OpenSeperator_action:
ST03_564_Y71_0.MoveInit:=TRUE;		(*Zuführung 1 Vereinzler AST/GST *)
ST03_564_Y71_2.MoveInit:=TRUE;		(*Zuführung 2 Vereinzler AST/GST *)
END_ACTION

ACTION WaitForPart_entry:
ProcessMessage02:='';
Delay(IN:=FALSE);
END_ACTION

ACTION WaitForPart_action:
ProcessMessage02:='2IM6';						(*warte auf Teil Übergabeposition 1*)
END_ACTION

ACTION WaitForPart_exit:
ProcessMessage02:='';
END_ACTION

ACTION CloseSeperator_action:
ST03_564_Y71_0.MoveWork:=TRUE;		(*Zuführung 1 Vereinzler AST/GST *)
ST03_564_Y71_2.MoveWork:=TRUE;		(*Zuführung 2 Vereinzler AST/GST *)
END_ACTION

ACTION OpenStopper_action:
IF 	NOT ST03_562_B67_7.BitInToCheck THEN	(*Zuführung 1 ISK auf Übergabepos. Robi*)
	ST03_564_Y71_1.MoveWork:=TRUE;		(*Zuführung 1 Stopper AST/GST *)
END_IF
IF 	NOT ST03_563_B70_7.BitInToCheck THEN	 (*Zuführung 2 ISK auf Übergabepos. Robi*)
	ST03_564_Y71_3.MoveWork:=TRUE;		(*Zuführung 2 Stopper AST/GST *)
END_IF
END_ACTION

ACTION WaitForPartOnPos1_entry:
ProcessMessage02:='';
Delay(IN:=FALSE);
END_ACTION

ACTION WaitForPartOnPos1_action:
ProcessMessage02:='2IM6';						(*warte auf Teil Übergabeposition 1*)
END_ACTION

ACTION WaitForPartOnPos1_exit:
ProcessMessage02:='';
END_ACTION

ACTION CloseStopper_action:
ST03_564_Y71_1.MoveInit:=TRUE;		(*Zuführung 1 Stopper AST/GST *)
ST03_564_Y71_3.MoveInit:=TRUE;		(*Zuführung 2 Stopper AST/GST *)
END_ACTION

ACTION OpenSeperator__action:
IF	NOT ST03_562_B69_6.BitInToCheck	THEN 	(*  ISK 1 anwesend am Stopper*)
	ST03_564_Y71_0.MoveInit:=TRUE;			(*Zuführung 1 Vereinzler AST/GST *)
END_IF
IF	NOT ST03_563_B70_6.BitInToCheck	THEN	 (*  ISK 2 anwesend am Stopper*)
	ST03_564_Y71_2.MoveInit:=TRUE;			(*Zuführung 2 Vereinzler AST/GST *)
END_IF
END_ACTION

ACTION SeqEnd_action:
SFCTime:=TIME_TO_DINT(TIME()-SFCTimeStart);
State:=STATE_WAIT;
END_ACTION

TRANSITION .ActualArea:
Robot01.ActualArea <> 4
END_TRANSITION

TRANSITION Check_Part:
NOT ST03_513_B70_7.BitInToCheck OR	(* ISK auf Übergabeposition  1*)
NOT ST03_514_B71_2.BitInToCheck OR	(* ISK auf Übergabeposition  2*)
NOT ST03_514_B71_5.BitInToCheck OR	(* ISK auf Übergabeposition  3*)
NOT ST03_514_B71_6.BitInToCheck		(* ISK auf Übergabeposition  4*)
END_TRANSITION

TRANSITION PosEmpty:
NOT ST03_562_B69_6.BitInToCheck	OR	 	(*  ISK 1 anwesend am Stopper*)
NOT ST03_563_B70_6.BitInToCheck		 	(*  ISK 2 anwesend am Stopper*)
END_TRANSITION

TRANSITION State Ok:
ST03_564_Y71_0.State=STATE_OK AND	(*Zuführung 1 Vereinzler AST/GST *)
ST03_564_Y71_2.State=STATE_OK 		(*Zuführung 2 Vereinzler AST/GST *)
END_TRANSITION

TRANSITION Part Ready:
ST03_562_B69_6.BitInToCheck	AND	(*  ISK 1 anwesend am Stopper*)
ST03_563_B70_6.BitInToCheck		 	(*  ISK 2 anwesend am Stopper*)
END_TRANSITION

TRANSITION PosFull:
ST03_562_B69_6.BitInToCheck	AND	 	(*  ISK 1 anwesend am Stopper*)
ST03_563_B70_6.BitInToCheck			 	(*  ISK 2 anwesend am Stopper*)
END_TRANSITION

TRANSITION State Ok:
ST03_564_Y71_0.State=STATE_OK AND	(*Zuführung 1 Vereinzler AST/GST *)
ST03_564_Y71_2.State=STATE_OK 		(*Zuführung 2 Vereinzler AST/GST *)
END_TRANSITION

TRANSITION Pos1o2_Empty:
NOT ST03_562_B67_7.BitInToCheck OR	(*Zuführung 1 ISK auf Übergabepos. Robi*)
NOT ST03_563_B70_7.BitInToCheck	 	(*Zuführung 2 ISK auf Übergabepos. Robi*)
END_TRANSITION

TRANSITION State Ok:
ST03_564_Y71_1.State=STATE_OK AND 	(*Zuführung 1 Stopper AST/GST *)
ST03_564_Y71_3.State=STATE_OK 		(*Zuführung 2 Stopper AST/GST *)
END_TRANSITION

TRANSITION Pos1and2 Ready:
ST03_562_B67_7.BitInToCheck 	AND	 (*Zuführung 1 ISK auf Übergabepos. Robi*)
ST03_563_B70_7.BitInToCheck 			 (*Zuführung 2 ISK auf Übergabepos. Robi*)
END_TRANSITION

TRANSITION Pos1and2Full:
ST03_562_B67_7.BitInToCheck AND	(*Zuführung 1 ISK auf Übergabepos. Robi*)
ST03_563_B70_7.BitInToCheck	 	(*Zuführung 2 ISK auf Übergabepos. Robi*)
END_TRANSITION

TRANSITION State Ok:
ST03_564_Y71_1.State=STATE_OK 	AND	(*Zuführung 1 Stopper AST/GST *)
ST03_564_Y71_3.State=STATE_OK 		(*Zuführung 2 Stopper AST/GST *)
END_TRANSITION
END_PROGRAM

(* POU Stations/ST_03_Ruestsaetze/ST_03_SFCs/Zufuehrungen/ST03_268_RP_Wendeeinheit, SFC *)
 PROGRAM ST03_268_RP_Wendeeinheit

VAR_OUTPUT
	SFCCurrentPOU			: STRING:='ST03_268_RP_Wendeeinheit';
	SFCCurrentStep			: STRING:='';
	FB_CurrentStepHistorie	: FB_CurrentStepHistorie;
	SFCTime					: DINT;
	State   				: StateObject	:= STATE_WAIT;
	Result  				: StateResult;

END_VAR
VAR_INPUT
	Start				:BOOL;
END_VAR
VAR
	MsgOK				: BOOL;
	MsgCancel			: BOOL;
	SFCRun				: BOOL;
	SFCTimeStart		: TIME;
	Delay				: TON;
	(* Userdefinded area *)
	WenderDone			: BOOL;
	OverrideHelp			:DINT;
END_VAR
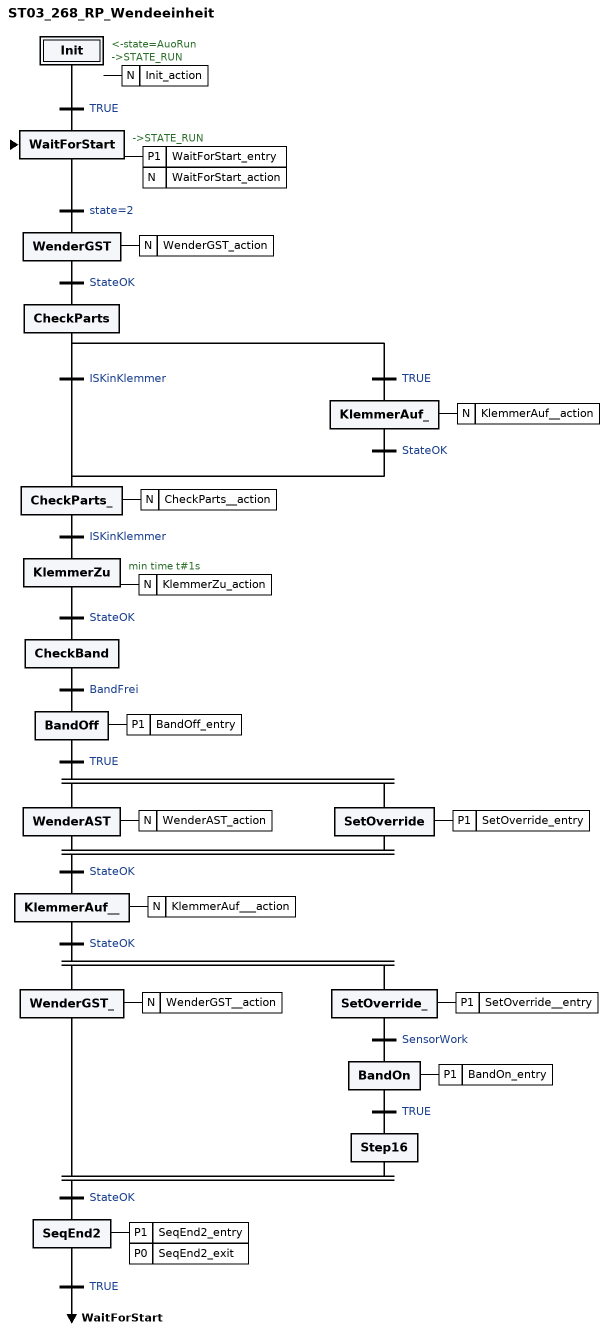
INITIAL_STEP Init: (* <-state=AuoRun / ->STATE_RUN *)
	Init_action(N);
END_STEP
TRANSITION FROM Init TO WaitForStart := TRUE;
END_TRANSITION
STEP WaitForStart: (* ->STATE_RUN *)
	WaitForStart_entry(P1);
	WaitForStart_action(N);
END_STEP
TRANSITION FROM WaitForStart TO WenderGST := state=2;
END_TRANSITION
STEP WenderGST:
	WenderGST_action(N);
END_STEP
TRANSITION FROM WenderGST TO CheckParts := StateOK;
END_TRANSITION
STEP CheckParts:
END_STEP
TRANSITION FROM CheckParts TO CheckParts_ := ISKinKlemmer;
END_TRANSITION
TRANSITION FROM CheckParts TO KlemmerAuf_ := TRUE;
END_TRANSITION
STEP KlemmerAuf_:
	KlemmerAuf__action(N);
END_STEP
TRANSITION FROM KlemmerAuf_ TO CheckParts_ := StateOK;
END_TRANSITION
STEP CheckParts_:
	CheckParts__action(N);
END_STEP
TRANSITION FROM CheckParts_ TO KlemmerZu := ISKinKlemmer;
END_TRANSITION
STEP KlemmerZu: (* min time t#1s *)
	KlemmerZu_action(N);
END_STEP
TRANSITION FROM KlemmerZu TO CheckBand := StateOK;
END_TRANSITION
STEP CheckBand:
END_STEP
TRANSITION FROM CheckBand TO BandOff := BandFrei;
END_TRANSITION
STEP BandOff:
	BandOff_entry(P1);
END_STEP
TRANSITION FROM BandOff TO (WenderAST, SetOverride) := TRUE;
END_TRANSITION
STEP WenderAST:
	WenderAST_action(N);
END_STEP
STEP SetOverride:
	SetOverride_entry(P1);
END_STEP
TRANSITION FROM (WenderAST, SetOverride) TO KlemmerAuf__ := StateOK;
END_TRANSITION
STEP KlemmerAuf__:
	KlemmerAuf___action(N);
END_STEP
TRANSITION FROM KlemmerAuf__ TO (WenderGST_, SetOverride_) := StateOK;
END_TRANSITION
STEP WenderGST_:
	WenderGST__action(N);
END_STEP
STEP SetOverride_:
	SetOverride__entry(P1);
END_STEP
TRANSITION FROM SetOverride_ TO BandOn := SensorWork;
END_TRANSITION
STEP BandOn:
	BandOn_entry(P1);
END_STEP
TRANSITION FROM BandOn TO Step16 := TRUE;
END_TRANSITION
STEP Step16:
END_STEP
TRANSITION FROM (WenderGST_, Step16) TO SeqEnd2 := StateOK;
END_TRANSITION
STEP SeqEnd2:
	SeqEnd2_entry(P1);
	SeqEnd2_exit(P0);
END_STEP
TRANSITION FROM SeqEnd2 TO WaitForStart := TRUE;
END_TRANSITION

ACTION Init_action:
Start:=FALSE;
State:=STATE_WAIT;
MsgOK:=FALSE;
MsgCancel:=FALSE;
SFCRun:=FALSE;
Result:=RESULT_NON;
IF 	OverrideHelp <> 0 THEN
	MP.ST02.Override_Band:=OverrideHelp;
END_IF

ST03_Band.bLockBand := FALSE;
END_ACTION

ACTION WaitForStart_entry:
;
END_ACTION

ACTION WaitForStart_action:
IF 	Start   THEN
	State:=STATE_RUN;
	Result:=RESULT_NON;
	SFCTimeStart:=TIME();
	Start:=FALSE;
	WenderDone:=FALSE;
ELSE
	State:=STATE_WAIT;
	MsgOK:=FALSE;
	MsgCancel:=FALSE;
	SFCRun:=FALSE;
END_IF
END_ACTION

ACTION WenderGST_action:
ST03_564_Y71_5.MoveInit:=TRUE;		(* Rinne schwenkern AST/GST *)
END_ACTION

ACTION KlemmerAuf__action:
ST03_564_Y71_4.MoveInit:=TRUE;		(* ISK Klemmer AST/GST *)
END_ACTION

ACTION CheckParts__action:
ProcessMessage01:='1IM6';						(*'warte auf Teil in Vereinzelung*)
END_ACTION

ACTION KlemmerZu_action:
ST03_564_Y71_4.MoveWork:=TRUE;		(* ISK Klemmer AST/GST *)
END_ACTION

ACTION BandOff_entry:
ST03_Band.bLockBand := TRUE;
END_ACTION

ACTION WenderAST_action:
ST03_564_Y71_5.MoveWork:=TRUE;		(* Rinne schwenkern AST/GST *)
END_ACTION

ACTION SetOverride_entry:
IF 	MP.ST02.Override_Band > 20 THEN
	OverrideHelp:=MP.ST02.Override_Band;
	MP.ST02.Override_Band:= 15;
END_IF
END_ACTION

ACTION KlemmerAuf___action:
ST03_564_Y71_4.MoveInit:=TRUE;	(* ISK Klemmer AST/GST *)
END_ACTION

ACTION WenderGST__action:
ST03_564_Y71_5.MoveInit:=TRUE;		(* Rinne schwenkern AST/GST *)
END_ACTION

ACTION SetOverride__entry:
MP.ST02.Override_Band:=OverrideHelp;
END_ACTION

ACTION BandOn_entry:
ST03_Band.bLockBand := FALSE;
END_ACTION

ACTION SeqEnd2_entry:
WenderDone:=TRUE;
END_ACTION

ACTION SeqEnd2_exit:
WenderDone:=FALSE;
END_ACTION

TRANSITION StateOK:
ST03_564_Y71_5.State = STATE_OK 	(* Rinne schwenkern AST/GST *)
END_TRANSITION

TRANSITION ISKinKlemmer:
ST03_565_B72_0.BitInToCheck AND	(* ISK 1 in Klemmer *)
ST03_565_B72_1.BitInToCheck 		(* ISK 2 in Klemmer *)
END_TRANSITION

TRANSITION StateOK:
ST03_564_Y71_4.State = STATE_OK		(*   ISK Klemmer AST/GST *)
END_TRANSITION

TRANSITION ISKinKlemmer:
ST03_565_B72_0.BitInToCheck AND 	(* ISK 1 in Klemmer *)
ST03_565_B72_1.BitInToCheck AND 	(* ISK 2 in Klemmer *)
(ST00_73_K4.BitInToCheck 	OR ST02_S1_40K01.BitInToCheck)		(*Schnittstelle Freigabe von Spritzmaschine (nur für Anlagen ohne Rundtisch)*)
END_TRANSITION

TRANSITION StateOK:
ST03_564_Y71_4.State = STATE_OK			(* ISK Klemmer AST/GST *)
END_TRANSITION

TRANSITION BandFrei:
ST03_562_B69_0.BitInToCheck  AND	(*Zuführung 1 frei zum schwenken*)
ST03_563_B70_0.BitInToCheck 	 	(*Zuführung 2 frei zum schwenken*)
END_TRANSITION

TRANSITION StateOK:
ST03_564_Y71_5.State = STATE_OK 	(* Förderband  Zuführung Vereinzelner Wender AST/GST *)
END_TRANSITION

TRANSITION StateOK:
ST03_564_Y71_4.State = STATE_OK	(* ISK Klemmer AST/GST *)
END_TRANSITION

TRANSITION SensorWork:
NOT ST03_564_Y71_5.SensorWorkIn[1].SensorSignal
END_TRANSITION

TRANSITION StateOK:
ST03_564_Y71_5.State = STATE_OK 	(* Rinne schwenkern AST/GST *)
END_TRANSITION
END_PROGRAM

(* POU Stations/ST_03_Ruestsaetze/ST_03_SFCs/Zufuehrungen/ST03_91pol_Zufuehrung, SFC *)
 PROGRAM ST03_91pol_Zufuehrung
VAR_OUTPUT
	SFCCurrentPOU		: STRING:='ST03_21pol_Zufuehrung';
	SFCCurrentStep		: STRING:='';
	FB_CurrentStepHistorie: FB_CurrentStepHistorie;
	SFCTime				: DINT;
	State   			: StateObject	:= STATE_WAIT;
	Result  			: StateResult;
END_VAR
VAR_INPUT
	Start				:BOOL;
END_VAR
VAR
	MsgOK				: BOOL;
	MsgCancel			: BOOL;
	SFCRun				: BOOL;
	SFCTimeStart		: TIME;
	Delay				: TON;
	(* Userdefinded area *)

END_VAR
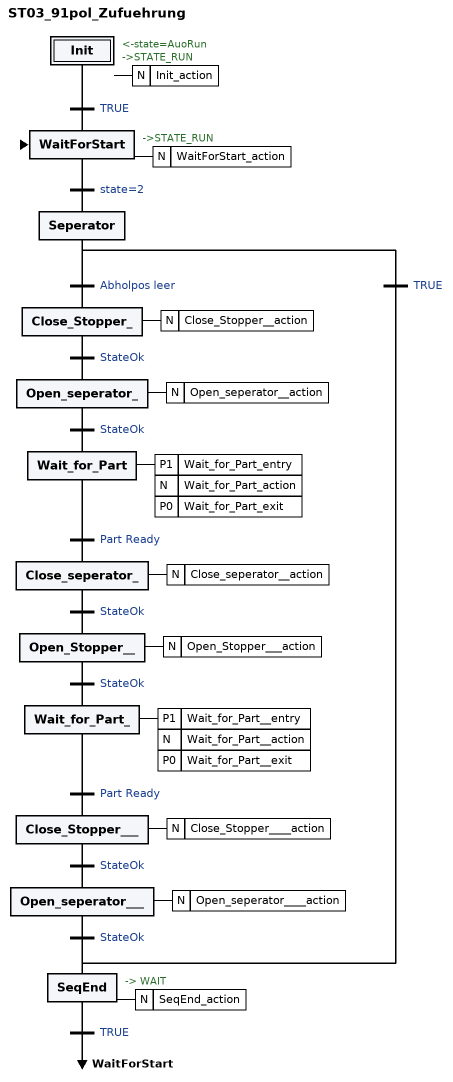
INITIAL_STEP Init: (* <-state=AuoRun / ->STATE_RUN *)
	Init_action(N);
END_STEP
TRANSITION FROM Init TO WaitForStart := TRUE;
END_TRANSITION
STEP WaitForStart: (* ->STATE_RUN *)
	WaitForStart_action(N);
END_STEP
TRANSITION FROM WaitForStart TO Seperator := state=2;
END_TRANSITION
STEP Seperator:
END_STEP
TRANSITION FROM Seperator TO Close_Stopper_ := Abholpos leer;
END_TRANSITION
TRANSITION FROM Seperator TO SeqEnd := TRUE;
END_TRANSITION
STEP Close_Stopper_:
	Close_Stopper__action(N);
END_STEP
TRANSITION FROM Close_Stopper_ TO Open_seperator_ := StateOk;
END_TRANSITION
STEP Open_seperator_:
	Open_seperator__action(N);
END_STEP
TRANSITION FROM Open_seperator_ TO Wait_for_Part := StateOk;
END_TRANSITION
STEP Wait_for_Part:
	Wait_for_Part_entry(P1);
	Wait_for_Part_action(N);
	Wait_for_Part_exit(P0);
END_STEP
TRANSITION FROM Wait_for_Part TO Close_seperator_ := Part Ready;
END_TRANSITION
STEP Close_seperator_:
	Close_seperator__action(N);
END_STEP
TRANSITION FROM Close_seperator_ TO Open_Stopper__ := StateOk;
END_TRANSITION
STEP Open_Stopper__:
	Open_Stopper___action(N);
END_STEP
TRANSITION FROM Open_Stopper__ TO Wait_for_Part_ := StateOk;
END_TRANSITION
STEP Wait_for_Part_:
	Wait_for_Part__entry(P1);
	Wait_for_Part__action(N);
	Wait_for_Part__exit(P0);
END_STEP
TRANSITION FROM Wait_for_Part_ TO Close_Stopper___ := Part Ready;
END_TRANSITION
STEP Close_Stopper___:
	Close_Stopper____action(N);
END_STEP
TRANSITION FROM Close_Stopper___ TO Open_seperator___ := StateOk;
END_TRANSITION
STEP Open_seperator___:
	Open_seperator____action(N);
END_STEP
TRANSITION FROM Open_seperator___ TO SeqEnd := StateOk;
END_TRANSITION
STEP SeqEnd: (* -> WAIT *)
	SeqEnd_action(N);
END_STEP
TRANSITION FROM SeqEnd TO WaitForStart := TRUE;
END_TRANSITION

ACTION Init_action:
Start:=FALSE;
State:=STATE_WAIT;
MsgOK:=FALSE;
MsgCancel:=FALSE;
SFCRun:=FALSE;
Result:=RESULT_NON;
END_ACTION

ACTION WaitForStart_action:
IF 	Start   THEN
	State:=STATE_RUN;
	Result:=RESULT_NON;
	SFCTimeStart:=TIME();
	Start:=FALSE;
ELSE
	State:=STATE_WAIT;
	MsgOK:=FALSE;
	MsgCancel:=FALSE;
	SFCRun:=FALSE;
END_IF
END_ACTION

ACTION Close_Stopper__action:
ST08_412_Y55_2.MoveWork:=TRUE;
END_ACTION

ACTION Open_seperator__action:
ST08_412_Y55_0.MoveInit:=TRUE;
END_ACTION

ACTION Wait_for_Part_entry:
ProcessMessage01:='';
Delay.IN:=FALSE;
Delay();
END_ACTION

ACTION Wait_for_Part_action:
ProcessMessage01:='1IM9';(*warte auf Teil in Stopper*)
Delay.IN:=ST08_412_B58_7.BitInToCheck;	(*  ISK an stopper.*)
Delay.PT:=T#50ms;
Delay();
END_ACTION

ACTION Wait_for_Part_exit:
ProcessMessage01:='';
END_ACTION

ACTION Close_seperator__action:
ST08_412_Y55_0.MoveWork:=TRUE;
END_ACTION

ACTION Open_Stopper___action:
ST08_412_Y55_2.MoveInit:=TRUE;
END_ACTION

ACTION Wait_for_Part__entry:
ProcessMessage01:='';
Delay.IN:=FALSE;
Delay();
END_ACTION

ACTION Wait_for_Part__action:
ProcessMessage01:='1IM10';(*warte auf Teil in Abholposition*)
Delay.IN:=	ST03_Init_AbholPos.RoboPos31 OR
			ST03_Init_AbholPos.RoboPos35;
Delay.PT:=T#50ms;
Delay();
END_ACTION

ACTION Wait_for_Part__exit:
ProcessMessage01:='';
END_ACTION

ACTION Close_Stopper____action:
ST08_412_Y55_2.MoveWork:=TRUE;
END_ACTION

ACTION Open_seperator____action:
ST08_412_Y55_0.MoveInit:=TRUE;
END_ACTION

ACTION SeqEnd_action:
SFCTime:=TIME_TO_DINT(TIME()-SFCTimeStart);
State:=STATE_WAIT;
END_ACTION

TRANSITION Abholpos leer:
NOT ST08_412_B59_0.BitInToCheck 		 (* Teil auf Abholpos *)
END_TRANSITION

TRANSITION StateOk:
ST08_412_Y55_2.State=STATE_OK
END_TRANSITION

TRANSITION StateOk:
ST08_412_Y55_0.State=STATE_OK
END_TRANSITION

TRANSITION Part Ready:
Delay.Q AND
Robot01.ActualArea <> 4
END_TRANSITION

TRANSITION StateOk:
ST08_412_Y55_0.State=STATE_OK
END_TRANSITION

TRANSITION StateOk:
ST08_412_Y55_2.State=STATE_OK
END_TRANSITION

TRANSITION Part Ready:
Delay.Q AND
Robot01.ActualArea <> 4
END_TRANSITION

TRANSITION StateOk:
ST08_412_Y55_2.State=STATE_OK
END_TRANSITION

TRANSITION StateOk:
ST08_412_Y55_0.State=STATE_OK
END_TRANSITION
END_PROGRAM

(* POU Stations/ST_03_Ruestsaetze/ST_03_SFCs/Zufuehrungen/ST03_33pol_Zufuehrung, SFC *)
 PROGRAM ST03_33pol_Zufuehrung
VAR_OUTPUT
	SFCCurrentPOU			: STRING:='ST03_33pol_Zufuehrung';
	SFCCurrentStep			: STRING:='';
	FB_CurrentStepHistorie:FB_CurrentStepHistorie;
	SFCTime					: DINT;
	State   				: StateObject	:= STATE_WAIT;
	Result  				: StateResult;
END_VAR
VAR_INPUT
	Start					:BOOL;
END_VAR
VAR
	MsgOK				: BOOL;
	MsgCancel			: BOOL;
	SFCRun				: BOOL;
	SFCTimeStart		: TIME;
	Delay				: TON;
	(* Userdefinded area *)

END_VAR
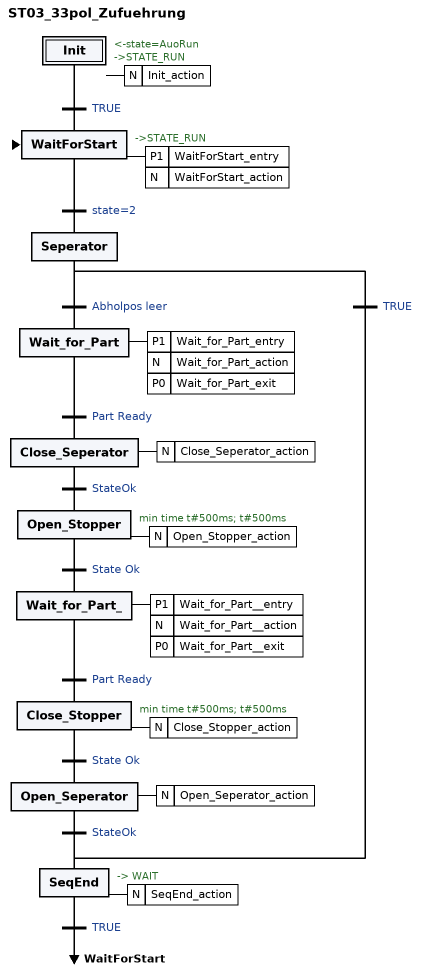
INITIAL_STEP Init: (* <-state=AuoRun / ->STATE_RUN *)
	Init_action(N);
END_STEP
TRANSITION FROM Init TO WaitForStart := TRUE;
END_TRANSITION
STEP WaitForStart: (* ->STATE_RUN *)
	WaitForStart_entry(P1);
	WaitForStart_action(N);
END_STEP
TRANSITION FROM WaitForStart TO Seperator := state=2;
END_TRANSITION
STEP Seperator:
END_STEP
TRANSITION FROM Seperator TO Wait_for_Part := Abholpos leer;
END_TRANSITION
TRANSITION FROM Seperator TO SeqEnd := TRUE;
END_TRANSITION
STEP Wait_for_Part:
	Wait_for_Part_entry(P1);
	Wait_for_Part_action(N);
	Wait_for_Part_exit(P0);
END_STEP
TRANSITION FROM Wait_for_Part TO Close_Seperator := Part Ready;
END_TRANSITION
STEP Close_Seperator:
	Close_Seperator_action(N);
END_STEP
TRANSITION FROM Close_Seperator TO Open_Stopper := StateOk;
END_TRANSITION
STEP Open_Stopper: (* min time t#500ms; t#500ms *)
	Open_Stopper_action(N);
END_STEP
TRANSITION FROM Open_Stopper TO Wait_for_Part_ := State Ok;
END_TRANSITION
STEP Wait_for_Part_:
	Wait_for_Part__entry(P1);
	Wait_for_Part__action(N);
	Wait_for_Part__exit(P0);
END_STEP
TRANSITION FROM Wait_for_Part_ TO Close_Stopper := Part Ready;
END_TRANSITION
STEP Close_Stopper: (* min time t#500ms; t#500ms *)
	Close_Stopper_action(N);
END_STEP
TRANSITION FROM Close_Stopper TO Open_Seperator := State Ok;
END_TRANSITION
STEP Open_Seperator:
	Open_Seperator_action(N);
END_STEP
TRANSITION FROM Open_Seperator TO SeqEnd := StateOk;
END_TRANSITION
STEP SeqEnd: (* -> WAIT *)
	SeqEnd_action(N);
END_STEP
TRANSITION FROM SeqEnd TO WaitForStart := TRUE;
END_TRANSITION

ACTION Init_action:
Start:=FALSE;
State:=STATE_WAIT;
MsgOK:=FALSE;
MsgCancel:=FALSE;
SFCRun:=FALSE;
Result:=RESULT_NON;
END_ACTION

ACTION WaitForStart_entry:
State:=STATE_OK;
END_ACTION

ACTION WaitForStart_action:
IF 	Start   THEN
	State:=STATE_RUN;
	Result:=RESULT_NON;
	SFCTimeStart:=TIME();
	Start:=FALSE;
ELSE
	State:=STATE_WAIT;
	MsgOK:=FALSE;
	MsgCancel:=FALSE;
	SFCRun:=FALSE;
END_IF
END_ACTION

ACTION Wait_for_Part_entry:
ProcessMessage01:='';
Delay.IN:=FALSE;
Delay();
END_ACTION

ACTION Wait_for_Part_action:
State:=STATE_RUN;
ProcessMessage01:='1IM9';(*warte auf Teil in Stopper*)
Delay.IN:=ST03_571_B69_6.BitInToCheck; 		(*  ISK an stopper.*)
Delay.PT:=T#500ms;
Delay();
END_ACTION

ACTION Wait_for_Part_exit:
ProcessMessage01:='';
END_ACTION

ACTION Close_Seperator_action:
ST03_572_Y70_0.MoveWork:=TRUE;		(* Förderband  Zuführung Vereinzler AST/GST *)
END_ACTION

ACTION Open_Stopper_action:
ST03_572_Y70_1.MoveWork:=TRUE;		(* Förderband  Züführung Stopper AST/GST *)
END_ACTION

ACTION Wait_for_Part__entry:
ProcessMessage01:='';
Delay.IN:=FALSE;
Delay();
END_ACTION

ACTION Wait_for_Part__action:
ProcessMessage01:='1IM10';(*warte auf Teil in Abholposition*)
Delay.IN:=ST03_571_B69_7.BitInToCheck; 		 (* ISK auf Abholposition Robi *)
Delay.PT:=T#500ms;
Delay();
END_ACTION

ACTION Wait_for_Part__exit:
ProcessMessage01:='';
END_ACTION

ACTION Close_Stopper_action:
ST03_572_Y70_1.MoveInit:=TRUE;		(* Förderband  Züführung Stopper AST/GST *)
END_ACTION

ACTION Open_Seperator_action:
ST03_572_Y70_0.MoveInit:=TRUE;		(* Förderband  Zuführung Vereinzler AST/GST *)
END_ACTION

ACTION SeqEnd_action:
SFCTime:=TIME_TO_DINT(TIME()-SFCTimeStart);
State:=STATE_WAIT;
END_ACTION

TRANSITION Abholpos leer:
NOT  ST03_571_B69_7.BitInToCheck		(*  ISK auf Abholposition Robi*)
END_TRANSITION

TRANSITION Part Ready:
Delay.Q AND
NOT ST03_571_B69_7.BitInToCheck	AND		(*  ISK auf Abholposition Robi*)
ST03_571_B69_6.BitInToCheck	AND				(*  ISK anwesend am Stoper*)
Robot01.ActualArea <> 4
END_TRANSITION

TRANSITION StateOk:
ST03_572_Y70_0.State=STATE_OK 	(* Förderband  Zuführung Vereinzler AST/GST *)
END_TRANSITION

TRANSITION State Ok:
ST03_572_Y70_1.State=STATE_OK 	(* Förderband  Züführung Stopper AST/GST *)
END_TRANSITION

TRANSITION Part Ready:
Delay.Q AND
Robot01.ActualArea <> 4
END_TRANSITION

TRANSITION State Ok:
ST03_572_Y70_1.State=STATE_OK 	(* Förderband  Züführung Stopper AST/GST *)
END_TRANSITION

TRANSITION StateOk:
ST03_572_Y70_0.State=STATE_OK 	(* Förderband  Zuführung Vereinzler AST/GST *)
END_TRANSITION
END_PROGRAM

(* POU zLibrary/ept/Service/_CallInit, ST *)
PROGRAM _CallInit


VAR



END_VAR
ST00_Init();
ST02_Init();
ST03_Init();

ST08_Init();
END_PROGRAM

(* POU Stations/ST_00/ST00__Init/ST00_Init, ST *)
PROGRAM ST00_Init


VAR


END_VAR
(* ----------------------------------------------------------------------------------------- *)
(* 																				Sicherungen																				 *)
(* ----------------------------------------------------------------------------------------- *)

(* Init ST00_40_F1 Vorsicherungen Leistung iO (DigIn) *)
ST00_40_F1.sInit.InstName                :='ST00_40_F1';
ST00_40_F1.sInit.Description             :='Sicherungsmodul 24VDC iO';
ST00_40_F1.sInit.BitInName               :='-40_F1';
ST00_40_F1.sInit.HomePosSignal           :=1; (* 0: Signal=Low, 1: Signal=High, 2: always  *)
ST00_40_F1.sInit.MaxTime                 :=2000;
ST00_40_F1.sInit.EnableInEveryMode       :=TRUE;

(* ----------------------------------------------------------------------------------------- *)
(* 																				Sicherheit																							 *)
(* ----------------------------------------------------------------------------------------- *)
(* Init ST03_210_S1 Not-Aus 1 Anlage ausgelöst (DigIn) *)
ST03_210_S1.sInit.InstName               :='ST03_210_S1';
ST03_210_S1.sInit.Description            :='Not-Aus 1 Anlage ausgelöst';
ST03_210_S1.sInit.BitInName              :='-210_S1';
ST03_210_S1.sInit.HomePosSignal          :=0; (* 0: Signal=Low, 1: Signal=High, 2: always  *)
ST03_210_S1.sInit.MaxTime                :=10;
ST03_210_S1.sInit.EnableInEveryMode   	 :=TRUE;

(* Init ST08_210_S2 Not-Aus 2 Anlage ausgelöst (DigIn) *)
ST08_210_S2.sInit.InstName               :='ST08_210_S2';
ST08_210_S2.sInit.Description            :='Not-Aus 2 Anlage ausgelöst';
ST08_210_S2.sInit.BitInName              :='-210_S2';
ST08_210_S2.sInit.HomePosSignal          :=1; (* 0: Signal=Low, 1: Signal=High, 2: always  *)
ST08_210_S2.sInit.MaxTime                :=10;
ST08_210_S2.sInit.EnableInEveryMode   	 :=TRUE;

(* Init ST00_X4_16 Not-Halt 2 Tampondrucker (DigIn) *)
ST00_X4_16.sInit.InstName               :='ST00_X4_16';
ST00_X4_16.sInit.Description            :='Not-Halt 2 Tampondrucker ausgelöst';
ST00_X4_16.sInit.BitInName              :='-X_16';
ST00_X4_16.sInit.HomePosSignal          :=0; (* 0: Signal=Low, 1: Signal=High, 2: always  *)
ST00_X4_16.sInit.MaxTime                :=10;
ST00_X4_16.sInit.EnableInEveryMode   	  :=TRUE;

(* Init ST00_200_A1_A1 Not-Aus iO (DigIn) *)
ST00_200_A1_A1.sInit.InstName            :='ST00_200_A1_A1';
ST00_200_A1_A1.sInit.Description         :='Not-Aus iO';
ST00_200_A1_A1.sInit.BitInName           :='-200_A1:A1';
ST00_200_A1_A1.sInit.HomePosSignal       :=1; (* 0: Signal=Low, 1: Signal=High, 2: always  *)
ST00_200_A1_A1.sInit.MaxTime             :=2000;
ST00_200_A1_A1.sInit.EnableInEveryMode   :=TRUE;

(* Init ST00_220_S1 Schutztüre 1 geöffnet (DigIn) *)
ST00_220_S1.sInit.InstName               :='ST00_220_S1';
ST00_220_S1.sInit.Description            :='Schutztüre 1 geöffnet';
ST00_220_S1.sInit.BitInName              :='-220_S1'; 
ST00_220_S1.sInit.HomePosSignal          :=0; (* 0: Signal=Low, 1: Signal=High, 2: always  *) 
ST00_220_S1.sInit.MaxTime                :=10;
ST00_220_S1.sInit.EnableInEveryMode   	 :=TRUE;

(* Init ST00_220_S2 Schutztüre 2 geöffnet (DigIn) *)
ST00_220_S2.sInit.InstName               :='ST00_220_S2';
ST00_220_S2.sInit.Description            :='Schutztüre 1 geöffnet';
ST00_220_S2.sInit.BitInName              :='-220_S2';
ST00_220_S2.sInit.HomePosSignal          :=0; (* 0: Signal=Low, 1: Signal=High, 2: always  *)
ST00_220_S2.sInit.MaxTime                :=10;
ST00_220_S2.sInit.EnableInEveryMode   	 :=TRUE;

(* Init ST00_223_S2_E1 Schutztüre 1 geschlossen (DigIn) *)
ST00_230_S2_E1.sInit.InstName            :='ST00_230_S2_E1';
ST00_230_S2_E1.sInit.Description         :='Schutztüre 1 geschlossen';
ST00_230_S2_E1.sInit.BitInName           :='-230_S2:E1';
ST00_230_S2_E1.sInit.HomePosSignal       :=2;(* :=1 @@@ *) (* 0: Signal=Low, 1: Signal=High, 2: always  *)
ST00_230_S2_E1.sInit.MaxTime             :=10;
ST00_230_S2_E1.sInit.EnableInEveryMode   	 :=TRUE;

(* Init ST00_240_S1 Schutztüre 9 geschlossen (DigIn) *)
ST00_240_S1.sInit.InstName            :='ST00_240_S1';
ST00_240_S1.sInit.Description         :='Schutztüre 9 geschlossen';
ST00_240_S1.sInit.BitInName           :='-240_S1';
ST00_240_S1.sInit.HomePosSignal       :=2;(* :=1 @@@ *) (* 0: Signal=Low, 1: Signal=High, 2: always  *)
ST00_240_S1.sInit.MaxTime             :=2000;
ST00_240_S1.sInit.EnableInEveryMode   	 :=TRUE;

(* Init ST00_226_S1 Hubtüre 1 Schleuse Einlauf STN 8 geschlossen (DigIn) *)
ST00_226_S1.sInit.InstName               :='ST00_226_S1';
ST00_226_S1.sInit.Description            :='Hubtüre 1 Schleuse Einlauf STN 8 geschlossen';
ST00_226_S1.sInit.BitInName              :='+0-226_S1';
ST00_226_S1.sInit.HomePosSignal          :=2; (* 0: Signal=Low, 1: Signal=High, 2: always  *)
ST00_226_S1.sInit.MaxTime                :=2000;
ST00_226_S1.sInit.EnableInEveryMode   	 :=TRUE;

(* Init ST00_226_S2 Hubtüre 2 Schleuse Einlauf STN 8 geschlossen (DigIn) *)
ST00_226_S2.sInit.InstName               :='ST00_226_S2';
ST00_226_S2.sInit.Description            :='Hubtüre 2 Schleuse Einlauf STN 8 geschlossen';
ST00_226_S2.sInit.BitInName              :='+0-226_S2';
ST00_226_S2.sInit.HomePosSignal          :=2; (* 0: Signal=Low, 1: Signal=High, 2: always  *)
ST00_226_S2.sInit.MaxTime                :=3000;
ST00_226_S2.sInit.EnableInEveryMode   	 :=TRUE;

(* Init ST00_227_S1 Hubtüre 3 Schleuse Auslauf STN 8 geschlossen (DigIn) *) 
ST00_227_S1.sInit.InstName               :='ST00_227_S1';
ST00_227_S1.sInit.Description            :='Hubtüre 3 Schleuse Auslauf STN 8 geschlossen';
ST00_227_S1.sInit.BitInName              :='+0-227_S1';
ST00_227_S1.sInit.HomePosSignal          :=2; (* 0: Signal=Low, 1: Signal=High, 2: always  *)
ST00_227_S1.sInit.MaxTime                :=2000;
ST00_227_S1.sInit.EnableInEveryMode   	 :=TRUE;

(* Init ST00_227_S2 Hubtüre 4 Schleuse Auslauf STN 8 geschlossen (DigIn) *)
ST00_227_S2.sInit.InstName               :='ST00_227_S2';
ST00_227_S2.sInit.Description            :='Hubtüre 4 Schleuse Auslauf STN 8 geschlossen';
ST00_227_S2.sInit.BitInName              :='+0-227_S2';
ST00_227_S2.sInit.HomePosSignal          :=2; (* 0: Signal=Low, 1: Signal=High, 2: always  *)
ST00_227_S2.sInit.MaxTime                :=2000;
ST00_227_S2.sInit.EnableInEveryMode   	 :=TRUE;

(* Init ST00_229_S1 Schutztüre Einlauf Tray STN 8 geschlossen (DigIn) *)
ST00_229_S1.sInit.InstName               :='ST00_229_S1';
ST00_229_S1.sInit.Description            :='Schutztüre Einlauf Tray STN 8 geschlossen';
ST00_229_S1.sInit.BitInName              :='+0-229_S1';
ST00_229_S1.sInit.HomePosSignal          :=2; (* 0: Signal=Low, 1: Signal=High, 2: always  *)
ST00_229_S1.sInit.MaxTime                :=2000;
ST00_229_S1.sInit.EnableInEveryMode   	 :=TRUE;

(* Init ST00_230_S1 Schutztüre Einlauf Tray STN 8 geschlossen (DigIn) *)
ST00_230_S1.sInit.InstName               :='ST00_230_S1';
ST00_230_S1.sInit.Description            :='Schutztüre Auslauf Tray STN 8 geschlossen';
ST00_230_S1.sInit.BitInName              :='+0-230_S1';
ST00_230_S1.sInit.HomePosSignal          :=2; (* 0: Signal=Low, 1: Signal=High, 2: always  *)
ST00_230_S1.sInit.MaxTime                :=2000;
ST00_230_S1.sInit.EnableInEveryMode   	 :=TRUE;

(* Init ST00_231_S1 Schutztüre Panel / Rutsche STN 8 geschlossen (DigIn) *)
ST00_231_S1.sInit.InstName               :='ST00_231_S1';
ST00_231_S1.sInit.Description            :='Schutztüre Panel / Rutsche STN 8 geschlossen';
ST00_231_S1.sInit.BitInName              :='+0-231_S1';
ST00_231_S1.sInit.HomePosSignal          :=2; (* 0: Signal=Low, 1: Signal=High, 2: always  *)
ST00_231_S1.sInit.MaxTime                :=2000;
ST00_231_S1.sInit.EnableInEveryMode   	 :=TRUE;

(* Init ST00_232_S1 Schutztüre 8 Auslauf Trays STN 8 geschlossen (DigIn) *)
ST00_232_S1.sInit.InstName               :='ST00_232_S1';
ST00_232_S1.sInit.Description            :='Schutztüre 8 Auslauf Trays STN 8 geschlossen';
ST00_232_S1.sInit.BitInName              :='+0-232_S1';
ST00_232_S1.sInit.HomePosSignal          :=2; (* 0: Signal=Low, 1: Signal=High, 2: always  *)
ST00_232_S1.sInit.MaxTime                :=2000;
ST00_232_S1.sInit.EnableInEveryMode   	 :=TRUE;

(* Init ST00_170_Motorschutz (DigIn) *)
ST00_170_Motorschutz.sInit.InstName              :='ST00_170_Motorschutz';
ST00_170_Motorschutz.sInit.Description            :='Motorschutz';
ST00_170_Motorschutz.sInit.BitInName              :='+0-170_Motorschutz';
ST00_170_Motorschutz.sInit.HomePosSignal          :=1; (* 0: Signal=Low, 1: Signal=High, 2: always  *)
ST00_170_Motorschutz.sInit.MaxTime                :=2000;
ST00_170_Motorschutz.sInit.EnableInEveryMode   	 :=TRUE;

(* Init ST00_170_Thermokontakt (DigIn) *)
ST00_170_Thermokont.sInit.InstName              :='ST00_170_Thermokont';
ST00_170_Thermokont.sInit.Description            :='Thermokontakt';
ST00_170_Thermokont.sInit.BitInName              :='+0-170_Thermokont';
ST00_170_Thermokont.sInit.HomePosSignal          :=1; (* 0: Signal=Low, 1: Signal=High, 2: always  *)
ST00_170_Thermokont.sInit.MaxTime                :=2000;
ST00_170_Thermokont.sInit.EnableInEveryMode   	 :=TRUE;

(* Init ST00_228_S1 Hubtüre 4 Schleuse Auslauf STN 8 geschlossen (DigIn) *)
ST00_228_S1.sInit.InstName               :='ST00_228_S1';
ST00_228_S1.sInit.Description            :='Pallettierer in Position';
ST00_228_S1.sInit.BitInName              :='+0-228_S1';
ST00_228_S1.sInit.HomePosSignal          :=2; (* 0: Signal=Low, 1: Signal=High, 2: always  *)
ST00_228_S1.sInit.MaxTime                :=2000;
ST00_228_S1.sInit.EnableInEveryMode   	 :=TRUE;


(* Init ST00_71_X1_3 Schnittstelle Bedrucken Tinte JSK auf Übergabeposition (DigIn) *)
ST00_71_X1_3.sInit.InstName            :='ST00_71_X1_3';
ST00_71_X1_3.sInit.Description         :='Bedrucken Tinte JSK auf Übergabeposition';
ST00_71_X1_3.sInit.BitInName           :='-71_X1_3';
ST00_71_X1_3.sInit.HomePosSignal       :=2; (* 0: Signal=Low, 1: Signal=High, 2: always  *)
ST00_71_X1_3.sInit.MaxTime             :=2000;
ST00_71_X1_3.sInit.EnableInEveryMode   :=FALSE;

(* Init ST00_71_X1_4 Schnittstelle Bedrucken Tinte Druckstation betriebsbereit (DigIn) *)
ST00_71_X1_4.sInit.InstName            :='ST00_71_X1_4';
ST00_71_X1_4.sInit.Description         :='Bedrucken Tinte Druckstation betriebsbereit';
ST00_71_X1_4.sInit.BitInName           :='-71_X1_4';
ST00_71_X1_4.sInit.HomePosSignal       :=2; (* 0: Signal=Low, 1: Signal=High, 2: always  *)
ST00_71_X1_4.sInit.MaxTime             :=2000;
ST00_71_X1_4.sInit.EnableInEveryMode   :=FALSE;

(* Init ST00_72_X1_3 Schnittstelle Tampondrucker Teil in Abholposition (DigIn) *)(*Band Entnahmeposition 1*)
ST00_72_X1_3.sInit.InstName            :='ST00_72_X1_3';
ST00_72_X1_3.sInit.Description         :='Band Entnahmeposition 1';
ST00_72_X1_3.sInit.BitInName           :='-72_X1_3';
ST00_72_X1_3.sInit.HomePosSignal       :=2; (* 0: Signal=Low, 1: Signal=High, 2: always  *)
ST00_72_X1_3.sInit.MaxTime             :=2000;
ST00_72_X1_3.sInit.EnableInEveryMode   :=FALSE;

(* Init ST00_72_X1_8 Schnittstelle Tampondrucker Druck abgeschlossen (DigIn) *)
ST00_72_X1_8.sInit.InstName            :='ST00_72_X1_8';
ST00_72_X1_8.sInit.Description         :='Tampondrucker Druck abgeschlossen';
ST00_72_X1_8.sInit.BitInName           :='-72_X1_8';
ST00_72_X1_8.sInit.HomePosSignal       :=2; (* 0: Signal=Low, 1: Signal=High, 2: always  *)
ST00_72_X1_8.sInit.MaxTime             :=2000;
ST00_72_X1_8.sInit.EnableInEveryMode   :=FALSE;

(* Init ST00_292_S1_STOP Bedienstelle Produktion Stop (DigIn) *)
ST00_292_S1_STOP.sInit.InstName          :='ST00_292_S1_STOP';
ST00_292_S1_STOP.sInit.Description       :='Bedienstelle Produktion Stop';
ST00_292_S1_STOP.sInit.BitInName         :='-292_S1:STOP';
ST00_292_S1_STOP.sInit.HomePosSignal     :=2; (* 0: Signal=Low, 1: Signal=High, 2: always  *)
ST00_292_S1_STOP.sInit.MaxTime           :=2000;
ST00_292_S1_STOP.sInit.EnableInEveryMode   	 :=TRUE;

(* Init ST00_292_S2_START Bedienstelle Produktion Start (DigIn) *)
ST00_292_S2_START.sInit.InstName         :='ST00_292_S2_START';
ST00_292_S2_START.sInit.Description      :='Bedienstelle Produktion Start';
ST00_292_S2_START.sInit.BitInName        :='-292_S2:START';
ST00_292_S2_START.sInit.HomePosSignal    :=2; (* 0: Signal=Low, 1: Signal=High, 2: always  *)
ST00_292_S2_START.sInit.MaxTime          :=2000;
ST00_292_S2_START.sInit.EnableInEveryMode   	 :=TRUE;

(* Init ST00_292_S3_RESET Bedienstelle Produktion Start (DigIn) *)
ST00_292_S3_RESET.sInit.InstName         :='ST00_292_S3_RESET';
ST00_292_S3_RESET.sInit.Description      :='Bedienstelle Produktion Reset';
ST00_292_S3_RESET.sInit.BitInName        :='-292_S3:RESET';
ST00_292_S3_RESET.sInit.HomePosSignal    :=2; (* 0: Signal=Low, 1: Signal=High, 2: always  *)
ST00_292_S3_RESET.sInit.MaxTime          :=2000;
ST00_292_S3_RESET.sInit.EnableInEveryMode   	 :=TRUE;

(* Init ST00_350_B20_0 Druckschalter Wartungseinheit Hauptluft min.6 bar (DigIn) *)
ST00_350_B20_0.sInit.InstName            :='ST00_350_B20_0';
ST00_350_B20_0.sInit.Description         :='Druckschalter Wartungseinheit Hauptluft min.6 bar';
ST00_350_B20_0.sInit.BitInName           :='-350_B20.0';
ST00_350_B20_0.sInit.HomePosSignal       :=2; (* 0: Signal=Low, 1: Signal=High, 2: always  *)
ST00_350_B20_0.sInit.MaxTime             :=2000;
ST00_350_B20_0.sInit.EnableInEveryMode   :=TRUE;

(* Init 	ST00_245_V1		Verriegelung Schutztüren-Leuchte (DigOutIn) *)
ST00_245_V1.sInit.InstName           :='ST00_245_V1';
ST00_245_V1.sInit.Description        :='Verriegelung Schutztüren';
ST00_245_V1.sInit.BitOutName         :='-245-V1';
ST00_245_V1.sInit.BitInName          :='';
ST00_245_V1.sInit.HomePosOutput      :=2; (* 0: Signal=Low, 1: Signal=High, 2: always  *)
ST00_245_V1.sInit.MaxTime            :=2000;
ST00_245_V1.sInit.EnableInEveryMode  :=TRUE;

(* Init 	ST00_245_V2_START		Bedienstelle Start-Leuchte (DigOutIn) *)
ST00_245_V2_START.sInit.InstName         :='ST00_245_V2_START';
ST00_245_V2_START.sInit.Description      :='Bedienstelle Start-Leuchte';
ST00_245_V2_START.sInit.BitOutName       :='-245_V2:START';
ST00_245_V2_START.sInit.BitInName        :='';
ST00_245_V2_START.sInit.HomePosOutput    :=2; (* 0: Signal=Low, 1: Signal=High, 2: always  *)
ST00_245_V2_START.sInit.MaxTime          :=2000;
ST00_245_V2_START.sInit.EnableInEveryMode   	 :=TRUE;

(* Init 	ST00_245_V3_RESET		Bedienstelle Reset-Schutztüren-Leuchte (DigOutIn) *)
ST00_245_V3_RESET.sInit.InstName         :='ST00_245_V3_RESET';
ST00_245_V3_RESET.sInit.Description      :='Bedienstelle Reset-Leuchte';
ST00_245_V3_RESET.sInit.BitOutName       :='-245_V3:RESET';
ST00_245_V3_RESET.sInit.BitInName        :='';
ST00_245_V3_RESET.sInit.HomePosOutput    :=2; (* 0: Signal=Low, 1: Signal=High, 2: always  *)
ST00_245_V3_RESET.sInit.MaxTime          :=2000;
ST00_245_V3_RESET.sInit.EnableInEveryMode:=TRUE;

(* Init 	ST00_245_S1_STOP 	Bedienstelle Produktion Stop (DigIn) *)
ST00_245_S1_STOP.sInit.InstName          :='ST00_245_S1_STOP';
ST00_245_S1_STOP.sInit.Description       :='Bedienstelle Produktion Stop';
ST00_245_S1_STOP.sInit.BitInName         :='-245_S1:STOP';
ST00_245_S1_STOP.sInit.HomePosSignal     :=2; (* 0: Signal=Low, 1: Signal=High, 2: always  *)
ST00_245_S1_STOP.sInit.MaxTime           :=2000;
ST00_245_S1_STOP.sInit.EnableInEveryMode :=TRUE;

(* Init 	ST00_245_S2_START	Bedienstelle Produktion Start (DigIn) *)
ST00_245_S2_START.sInit.InstName         :='ST00_245_S2_START';
ST00_245_S2_START.sInit.Description      :='Bedienstelle Produktion Start';
ST00_245_S2_START.sInit.BitInName        :='-245_S2:START';
ST00_245_S2_START.sInit.HomePosSignal    :=2; (* 0: Signal=Low, 1: Signal=High, 2: always  *)
ST00_245_S2_START.sInit.MaxTime          :=2000;
ST00_245_S2_START.sInit.EnableInEveryMode:=TRUE;

(* Init 	ST00_245_S3_RESET	Bedienstelle Produktion Reset (DigIn) *)
ST00_245_S3_RESET.sInit.InstName         :='ST00_245_S3_RESET';
ST00_245_S3_RESET.sInit.Description      :='Bedienstelle Produktion Reset';
ST00_245_S3_RESET.sInit.BitInName        :='-245_S3:RESET';
ST00_245_S3_RESET.sInit.HomePosSignal    :=2; (* 0: Signal=Low, 1: Signal=High, 2: always  *)
ST00_245_S3_RESET.sInit.MaxTime			 :=2000;
ST00_245_S3_RESET.sInit.EnableInEveryMode:=TRUE;


(* ----------------------------------------------------------------------------------------- *)
(* 																			Ausgänge																						 *)
(* ----------------------------------------------------------------------------------------- *)

(* Init ST00_31_K1 Beleuchtung Anlage (DigOutIn) *)
ST00_31_K1.sInit.InstName                :='ST00_31_K1';
ST00_31_K1.sInit.Description             :='Beleuchtung Anlage';
ST00_31_K1.sInit.BitOutName              :='-31_K1'; 
ST00_31_K1.sInit.BitInName               :='';
ST00_31_K1.sInit.HomePosOutput           :=2; (* 0: Signal=Low, 1: Signal=High, 2: always  *)
ST00_31_K1.sInit.MaxTime                 :=2000;
ST00_31_K1.sInit.EnableInEveryMode   	 	:=TRUE;
ST00_31_K1.sInit.EnableVisuInEveryMode   :=TRUE;

(* Init ST00_350_H1 Signalsäule RD Maschine Alarm/Störung (DigOutIn) *)
ST00_350_H1.sInit.InstName               :='ST00_350_H1';
ST00_350_H1.sInit.Description            :='Signalsäule RD Maschine Alarm/Störung';
ST00_350_H1.sInit.BitOutName             :='-350_H1'; 
ST00_350_H1.sInit.BitInName              :=''; 
ST00_350_H1.sInit.HomePosOutput          :=2; (* 0: Signal=Low, 1: Signal=High, 2: always  *)
ST00_350_H1.sInit.MaxTime                :=2000;
ST00_350_H1.sInit.EnableInEveryMode   	 :=TRUE;

(* Init ST00_350_H2 Signalsäule YE Bedienereingriff erforderlich (DigOutIn) *)
ST00_350_H2.sInit.InstName               :='ST00_350_H2';
ST00_350_H2.sInit.Description            :='Signalsäule YE Bedienereingriff erforderlich';
ST00_350_H2.sInit.BitOutName             :='-350_H2';
ST00_350_H2.sInit.BitInName              :='';
ST00_350_H2.sInit.HomePosOutput          :=2; (* 0: Signal=Low, 1: Signal=High, 2: always  *)
ST00_350_H2.sInit.MaxTime                :=2000;
ST00_350_H2.sInit.EnableInEveryMode   	 :=TRUE;

(* Init ST00_350_H3 Signalsäule GN Maschine Automatik (DigOutIn) *)
ST00_350_H3.sInit.InstName               :='ST00_350_H3';
ST00_350_H3.sInit.Description            :='Signalsäule GN Maschine Automatik';
ST00_350_H3.sInit.BitOutName             :='-350_H3'; 
ST00_350_H3.sInit.BitInName              :=''; 
ST00_350_H3.sInit.HomePosOutput          :=2; (* 0: Signal=Low, 1: Signal=High, 2: always  *)
ST00_350_H3.sInit.MaxTime                :=2000;
ST00_350_H3.sInit.EnableInEveryMode   	 :=TRUE;

(* Init ST00_200_A1_E4 Quittierung Not-Aus (DigOutIn) *)
ST00_200_A1_E4.sInit.InstName            :='ST00_200_A1_E4';
ST00_200_A1_E4.sInit.Description         :='Quittierung Not-Aus';
ST00_200_A1_E4.sInit.BitOutName          :='-200_A1:E4'; 
ST00_200_A1_E4.sInit.BitInName           :=''; 
ST00_200_A1_E4.sInit.HomePosSignal       :=0; (* 0: Signal=Low, 1: Signal=High, 2: always  *)
ST00_200_A1_E4.sInit.MaxTime             :=2000;
ST00_200_A1_E4.sInit.EnableInEveryMode   :=TRUE;
ST00_200_A1_E4.sInit.EnableVisuInEveryMode :=TRUE;

(* Init ST00_220_S1_S31 Verriegelung Schutztüren (DigOutIn) *)
ST00_220_S1_S31.sInit.InstName           :='ST00_220_S1_S31';
ST00_220_S1_S31.sInit.Description        :='Verriegelung Schutztüren';
ST00_220_S1_S31.sInit.BitOutName         :='-220-S1:S31';
ST00_220_S1_S31.sInit.BitInName          :='';
ST00_220_S1_S31.sInit.HomePosOutput      :=2; (* 0: Signal=Low, 1: Signal=High, 2: always  *)
ST00_220_S1_S31.sInit.MaxTime            :=2000;
ST00_220_S1_S31.sInit.EnableInEveryMode   	 :=TRUE;

(* Init ST00_292_H2_START Bedienstelle Start-Leuchte (DigOutIn) *)
ST00_292_H2_START.sInit.InstName         :='ST00_292_H2_START';
ST00_292_H2_START.sInit.Description      :='Bedienstelle Start-Leuchte';
ST00_292_H2_START.sInit.BitOutName       :='-292_H2:START';
ST00_292_H2_START.sInit.BitInName        :='';
ST00_292_H2_START.sInit.HomePosOutput    :=2; (* 0: Signal=Low, 1: Signal=High, 2: always  *)
ST00_292_H2_START.sInit.MaxTime          :=2000;
ST00_292_H2_START.sInit.EnableInEveryMode   	 :=TRUE;

(* Init ST00_292_H3_RESET Bedienstelle Reset-Leuchte (DigOutIn) *)
ST00_292_H3_RESET.sInit.InstName         :='ST00_292_H3_RESET';
ST00_292_H3_RESET.sInit.Description      :='Bedienstelle Reset-Leuchte';
ST00_292_H3_RESET.sInit.BitOutName       :='-292_H3:RESET';
ST00_292_H3_RESET.sInit.BitInName        :='';
ST00_292_H3_RESET.sInit.HomePosOutput    :=2; (* 0: Signal=Low, 1: Signal=High, 2: always  *)
ST00_292_H3_RESET.sInit.MaxTime          :=2000;
ST00_292_H3_RESET.sInit.EnableInEveryMode   	 :=TRUE;

(* Init ST00_71_K2 Schnittstelle Bedrucken Tinte Abholposition frei (DigOutIn) *)
ST00_71_K2.sInit.InstName             :='ST00_71_K2';
ST00_71_K2.sInit.Description          :='Bedrucken Tinte Abholposition frei';
ST00_71_K2.sInit.BitOutName           :='-71_K1';
ST00_71_K2.sInit.BitInName            :='';
ST00_71_K2.sInit.HomePosSignal        :=2; (* 0: Signal=Low, 1: Signal=High, 2: always  *)
ST00_71_K2.sInit.HomePosOutput	 :=2; (* 0: Signal=Low, 1: Signal=High, 2: always  *)
ST00_71_K2.sInit.MaxTime              :=2000;
ST00_71_K2.sInit.EnableVisuInEveryMode:=TRUE;

(* Schnittstelle Förderband frei für Spritzmaschine(DigOutIn) *)
ST00_73_K3.sInit.InstName             :='ST00_73_K3';
ST00_73_K3.sInit.Description          :='Förderband frei für Spritzmaschine';
ST00_73_K3.sInit.BitOutName           :='-73_K3';
ST00_73_K3.sInit.BitInName            :='';
ST00_73_K3.sInit.HomePosSignal        :=2; (* 0: Signal=Low, 1: Signal=High, 2: always  *)
ST00_73_K3.sInit.HomePosOutput				:=2; (* 0: Signal=Low, 1: Signal=High, 2: always  *)
ST00_73_K3.sInit.MaxTime              :=2000;

(*ST00_73_K4  Schnittstelle Freigabe von Spritzmaschine (nur für Anlagen ohne Rundtisch) (DigIn)*)
ST00_73_K4.sInit.InstName                :='ST00_73_K4';
ST00_73_K4.sInit.Description             :=' Freigabe Spritzmaschine';
ST00_73_K4.sInit.BitInName               :='-73_K4';
ST00_73_K4.sInit.HomePosSignal   	 :=2; (* 0: Signal=Low, 1: Signal=High, 2: always  *)
ST00_73_K4.sInit.MaxTime                 :=2000;

(* Init ST00_74_B7_2 Stopper GST1 DS (ValveSensor) *)
ST00_74_B7_2.sInit.InstName            :='ST00_74_B7_2';
ST00_74_B7_2.sInit.BitName            :='+0_74_B7_2';
ST00_74_B7_2.sInit.Description         :='Stopper GST1 DS';
ST00_74_B7_2.sInit.SensorType          :=sValveSensorType_INIT;

(* Init ST00_74_B7_3 Stopper GST1 DS (ValveSensor) *)
ST00_74_B7_3.sInit.InstName            :='ST00_74_B7_3';
ST00_74_B7_3.sInit.BitName            :='+0_74_B7_3';
ST00_74_B7_3.sInit.Description         :='Stopper GST2 PS';
ST00_74_B7_3.sInit.SensorType          :=sValveSensorType_INIT;

(* Init ST00_74_B7_4 Vereinzeler AST1 DS (ValveSensor) *)
ST00_74_B7_4.sInit.InstName            :='ST00_74_B7_4';
ST00_74_B7_4.sInit.BitName            :='+0_74_B7_4';
ST00_74_B7_4.sInit.Description         :='Vereinzeler GST1 DS';
ST00_74_B7_4.sInit.SensorType          :=sValveSensorType_INIT;

(* Init ST00_74_B7_5 Vereinzeler AST2 PS (ValveSensor) *)
ST00_74_B7_5.sInit.InstName            :='ST00_74_B7_5';
ST00_74_B7_5.sInit.BitName            :='+0_74_B7_5';
ST00_74_B7_5.sInit.Description         :='Vereinzeler GST2 PS';
ST00_74_B7_5.sInit.SensorType          :=sValveSensorType_INIT;

(* Init ST00_74_B7_6  Vereinzeler GST1 DS(ValveSensor) *)
ST00_74_B7_6.sInit.InstName            :='ST00_74_B7_6';
ST00_74_B7_6.sInit.BitName            :='+0_74_B7_6';
ST00_74_B7_6.sInit.Description         :='Vereinzeler AST1 DS';
ST00_74_B7_6.sInit.SensorType          :=sValveSensorType_WORK;

(* Init ST00_74_B7_7 Vereinzeler GST2 PS (ValveSensor) *)
ST00_74_B7_7.sInit.InstName            :='ST00_74_B7_7';
ST00_74_B7_7.sInit.BitName            :='+0_74_B7_7';
ST00_74_B7_7.sInit.Description         :='Vereinzeler AST2 PS';
ST00_74_B7_7.sInit.SensorType          :=sValveSensorType_WORK;

(* Init ST00_74_Y2_4 Stopper ISK (lt. Schaltplan 62Y1)(Valve) *)
ST00_74_Y2_4.sInit.InstName            :='ST00_74_Y2_4';
ST00_74_Y2_4.sInit.BitName            :='+0_74_Y2_4';
ST00_74_Y2_4.sInit.Description         :='Stopper Bandstrecke';
ST00_74_Y2_4.sInit.HomePosDefine       :=HOME_ALWAYS;
ST00_74_Y2_4.sInit.InitDescription     :='GS';
ST00_74_Y2_4.sInit.WorkDescription     :='AS';
ST00_74_Y2_4.sInit.DampBothTime        :=200;
ST00_74_Y2_4.sInit.KindOfValve         :='A';
ST00_74_Y2_4.sInit.MaxTime             :=2000;

(* Init ST00_74_Y2_5 Vereinzeler ISK (lt. Schaltplan 62Y3)(Valve) *)
ST00_74_Y2_5.sInit.InstName            :='ST00_74_Y2_5';
ST00_74_Y2_5.sInit.BitName            :='+0_74_Y2_5';
ST00_74_Y2_5.sInit.Description         :='Vereinzeler Bandstrecke';
ST00_74_Y2_5.sInit.HomePosDefine       :=HOME_ALWAYS;
ST00_74_Y2_5.sInit.InitDescription     :='GS';
ST00_74_Y2_5.sInit.WorkDescription     :='AS';
ST00_74_Y2_5.sInit.DampBothTime        :=200;
ST00_74_Y2_5.sInit.KindOfValve         :='A';
ST00_74_Y2_5.sInit.MaxTime             :=2000;
END_PROGRAM

(* POU Stations/ST_02_RT_Tampondrucker/ST02__Init/ST02_Init, ST *)
PROGRAM ST02_Init


VAR


END_VAR
(* ----------------------------------------------------------------------------------------- *)

(* Init ST02_S1_6A01 ST02 Sicherung 24V  (DigIn) *)
ST02_S1_6A01.sInit.InstName                :='ST02_S1_6A01';
ST02_S1_6A01.sInit.Description             :='Sicherungsmodul 24VDC';
ST02_S1_6A01.sInit.BitInName               :='-S1_6A01';
ST02_S1_6A01.sInit.HomePosSignal   :=1; (* 0: Signal=Low, 1: Signal=High, 2: always  *)
ST02_S1_6A01.sInit.MaxTime                 :=2000;
ST02_S1_6A01.sInit.EnableInEveryMode       :=TRUE;

(* ----------------------------------------------------------------------------------------- *)
(* ----------------------------------------------------------------------------------------- *)
(* Init ST02_FDB_55X1_5_READY IFM Kamera Flügelerkennung links Ready (DigIn) *)
ST02_FDB_55X1_5_READY.sInit.InstName          :='ST02_FDB_55X1_5_READY';
ST02_FDB_55X1_5_READY.sInit.Description       :='IFM Kamera links ready';
ST02_FDB_55X1_5_READY.sInit.BitInName         :='+55X1_5_READY';
ST02_FDB_55X1_5_READY.sInit.HomePosSignal     :=2; (* 0: Signal=Low, 1: Signal=High, 2: always  *)
ST02_FDB_55X1_5_READY.sInit.MaxTime           :=2000;

(* Init ST02_FDB_55X1_6_IO IFM Kamera Flügelerkennung links Ergebnis iO (DigIn) *)
ST02_FDB_55X1_6_IO.sInit.InstName          :='ST02_FDB_55X1_6_IO';
ST02_FDB_55X1_6_IO.sInit.Description       :='IFM Kamera links Ergebnis iO';
ST02_FDB_55X1_6_IO.sInit.BitInName         :='+55X1_6_IO';
ST02_FDB_55X1_6_IO.sInit.HomePosSignal     :=2; (* 0: Signal=Low, 1: Signal=High, 2: always  *)
ST02_FDB_55X1_6_IO.sInit.MaxTime           :=2000;

(* Init ST02_FDB_55X1_6_NIO IFM Kamera Flügelerkennung links Ergebnis niO (DigIn) *)
ST02_FDB_55X1_6_NIO.sInit.InstName          :='ST02_FDB_55X1_6_NIO';
ST02_FDB_55X1_6_NIO.sInit.Description       :='IFM Kamera links Ergebnis niO';
ST02_FDB_55X1_6_NIO.sInit.BitInName         :='+55X1_6_NIO';
ST02_FDB_55X1_6_NIO.sInit.HomePosSignal     :=2; (* 0: Signal=Low, 1: Signal=High, 2: always  *)
ST02_FDB_55X1_6_NIO.sInit.MaxTime           :=2000;

(* Init ST02_FDB_55X1_2_TRIGGER IFM Kamera Flügelerkennung links Trigger (DigOutIn) *)
ST02_FDB_55X1_2_TRIGGER.sInit.InstName          :='ST02_FDB_55X1_2_TRIGGER';
ST02_FDB_55X1_2_TRIGGER.sInit.Description       :='IFM Kamera links Trigger';
ST02_FDB_55X1_2_TRIGGER.sInit.BitOutName        :='+55X1_2_TRIGGER';
ST02_FDB_55X1_2_TRIGGER.sInit.BitInName         :='';
ST02_FDB_55X1_2_TRIGGER.sInit.HomePosSignal     :=2; (* 0: Signal=Low, 1: Signal=High, 2: always  *)
ST02_FDB_55X1_2_TRIGGER.sInit.MaxTime           :=2000;

(* Init ST02_FDB_55X1_7_JOB_BIT1 IFM Kamera links Jobwechsel Bit1 (DigOutIn) *)
ST02_FDB_55X1_7_JOB_BIT1.sInit.InstName          :='ST02_FDB_55X1_7_JOB_BIT1';
ST02_FDB_55X1_7_JOB_BIT1.sInit.Description       :='IFM Kamera  Job Bit 1';
ST02_FDB_55X1_7_JOB_BIT1.sInit.BitOutName        :='+55X1_7_JOB_BIT1';
ST02_FDB_55X1_7_JOB_BIT1.sInit.BitInName         :='';
ST02_FDB_55X1_7_JOB_BIT1.sInit.HomePosSignal     :=2; (* 0: Signal=Low, 1: Signal=High, 2: always  *)
ST02_FDB_55X1_7_JOB_BIT1.sInit.MaxTime           :=2000;

(* Init ST02_FDB_55X1_7_JOB_BIT2 IFM Kamera links Jobwechsel Bit2 (DigOutIn) *)
ST02_FDB_55X1_7_JOB_BIT2.sInit.InstName          :='ST02_FDB_55X1_7_JOB_BIT2';
ST02_FDB_55X1_7_JOB_BIT2.sInit.Description       :='IFM Kamera  Job Bit 2';
ST02_FDB_55X1_7_JOB_BIT2.sInit.BitOutName        :='+55X1_7_JOB_BIT2';
ST02_FDB_55X1_7_JOB_BIT2.sInit.BitInName         :='';
ST02_FDB_55X1_7_JOB_BIT2.sInit.HomePosSignal     :=2; (* 0: Signal=Low, 1: Signal=High, 2: always  *)
ST02_FDB_55X1_7_JOB_BIT2.sInit.MaxTime           :=2000;
(* Init ST02_FDB_56X1_5_READY IFM Kamera Flügelerkennung rechts Ready (DigIn) *)
ST02_FDB_56X1_5_READY.sInit.InstName          :='ST02_FDB_56X1_5_READY';
ST02_FDB_56X1_5_READY.sInit.Description       :='IFM Kamera rechts ready';
ST02_FDB_56X1_5_READY.sInit.BitInName         :='+56X1_5_READY';
ST02_FDB_56X1_5_READY.sInit.HomePosSignal     :=2; (* 0: Signal=Low, 1: Signal=High, 2: always  *)
ST02_FDB_56X1_5_READY.sInit.MaxTime           :=2000;

(* Init ST02_FDB_56X1_6_IO IFM Kamera Flügelerkennung rechts Ergebnis iO (DigIn) *)
ST02_FDB_56X1_6_IO.sInit.InstName          :='ST02_FDB_56X1_6_IO';
ST02_FDB_56X1_6_IO.sInit.Description       :='IFM Kamera rechts Ergebnis iO';
ST02_FDB_56X1_6_IO.sInit.BitInName         :='+56X1_6_IO';
ST02_FDB_56X1_6_IO.sInit.HomePosSignal     :=2; (* 0: Signal=Low, 1: Signal=High, 2: always  *)
ST02_FDB_56X1_6_IO.sInit.MaxTime           :=2000;

(* Init ST02_FDB_56X1_6_NIO IFM Kamera Flügelerkennung rechts Ergebnis niO (DigIn) *)
ST02_FDB_56X1_6_NIO.sInit.InstName          :='ST02_FDB_56X1_6_NIO';
ST02_FDB_56X1_6_NIO.sInit.Description       :='IFM Kamera rechts Ergebnis niO';
ST02_FDB_56X1_6_NIO.sInit.BitInName         :='+56X1_6_NIO';
ST02_FDB_56X1_6_NIO.sInit.HomePosSignal     :=2; (* 0: Signal=Low, 1: Signal=High, 2: always  *)
ST02_FDB_56X1_6_NIO.sInit.MaxTime           :=2000;

(* Init ST02_FDB_56X1_2_TRIGGER IFM Kamera Flügelerkennung rechts Trigger (DigOutIn) *)
ST02_FDB_56X1_2_TRIGGER.sInit.InstName          :='ST02_FDB_56X1_2_TRIGGER';
ST02_FDB_56X1_2_TRIGGER.sInit.Description       :='IFM Kamera rechts Trigger';
ST02_FDB_56X1_2_TRIGGER.sInit.BitOutName        :='+56X1_2_TRIGGER';
ST02_FDB_56X1_2_TRIGGER.sInit.BitInName         :='';
ST02_FDB_56X1_2_TRIGGER.sInit.HomePosSignal     :=2; (* 0: Signal=Low, 1: Signal=High, 2: always  *)
ST02_FDB_56X1_2_TRIGGER.sInit.MaxTime           :=2000;

(* Init ST02_FDB_56X1_7_JOB_BIT1 IFM Kamera rechts Jobwechsel Bit1 (DigOutIn) *)
ST02_FDB_56X1_7_JOB_BIT1.sInit.InstName          :='ST02_FDB_56X1_7_JOB_BIT1';
ST02_FDB_56X1_7_JOB_BIT1.sInit.Description       :='IFM Kamera  Job Bit 1';
ST02_FDB_56X1_7_JOB_BIT1.sInit.BitOutName        :='+56X1_7_JOB_BIT1';
ST02_FDB_56X1_7_JOB_BIT1.sInit.BitInName         :='';
ST02_FDB_56X1_7_JOB_BIT1.sInit.HomePosSignal     :=2; (* 0: Signal=Low, 1: Signal=High, 2: always  *)
ST02_FDB_56X1_7_JOB_BIT1.sInit.MaxTime           :=2000;

(* Init ST02_FDB_56X1_7_JOB_BIT2 IFM Kamera rechts Jobwechsel Bit2 (DigOutIn) *)
ST02_FDB_56X1_7_JOB_BIT2.sInit.InstName          :='ST02_FDB_56X1_7_JOB_BIT2';
ST02_FDB_56X1_7_JOB_BIT2.sInit.Description       :='IFM Kamera  Job Bit 2';
ST02_FDB_56X1_7_JOB_BIT2.sInit.BitOutName        :='+56X1_7_JOB_BIT2';
ST02_FDB_56X1_7_JOB_BIT2.sInit.BitInName         :='';
ST02_FDB_56X1_7_JOB_BIT2.sInit.HomePosSignal     :=2; (* 0: Signal=Low, 1: Signal=High, 2: always  *)
ST02_FDB_56X1_7_JOB_BIT2.sInit.MaxTime           :=2000;

(* Init ST02_FDB_54_B41 Kamera ISK anwesend an Prüfposition (DigIn) *)
ST02_FDB_54_B41.sInit.InstName          :='ST02_FDB_54_B41';
ST02_FDB_54_B41.sInit.Description       :='Kamera ISK an Prüfposition';
ST02_FDB_54_B41.sInit.BitInName         :='+54B41';
ST02_FDB_54_B41.sInit.HomePosSignal     :=2; (* 0: Signal=Low, 1: Signal=High, 2: always  *)
ST02_FDB_54_B41.sInit.MaxTime           :=2000;

(* Init ST02_DT_65B11 Tampondrucker Nest 1 leer (DigIn) *)
ST02_DT_65B11.sInit.InstName            :='ST02_DT_65B11';
ST02_DT_65B11.sInit.Description         :='Tampondrucker Nest 1 leer';
ST02_DT_65B11.sInit.BitInName           :='+65B11';
ST02_DT_65B11.sInit.HomePosSignal       :=2; (* 0: Signal=Low, 1: Signal=High, 2: always  *)
ST02_DT_65B11.sInit.MaxTime             :=2000;
ST02_DT_65B11.sInit.EnableInEveryMode   :=FALSE;

(* Init ST02_DT_65B21 Tampondrucker Nest 2 leer (DigIn) *)
ST02_DT_65B21.sInit.InstName            :='ST02_DT_65B21';
ST02_DT_65B21.sInit.Description         :='Tampondrucker Nest 2 leer';
ST02_DT_65B21.sInit.BitInName           :='+65B21';
ST02_DT_65B21.sInit.HomePosSignal       :=2; (* 0: Signal=Low, 1: Signal=High, 2: always  *)
ST02_DT_65B21.sInit.MaxTime             :=2000;
ST02_DT_65B21.sInit.EnableInEveryMode   :=FALSE;

(* Init ST02_S1_70K61_A1 Start Bedruckung (DigOutIn) *)
ST02_S1_70K61_A1.sInit.InstName          :='ST02_S1_70K61_A1';
ST02_S1_70K61_A1.sInit.Description       :='Start Bedruckung';
ST02_S1_70K61_A1.sInit.BitOutName        :='+70K61_A1';
ST02_S1_70K61_A1.sInit.BitInName         :='';
ST02_S1_70K61_A1.sInit.HomePosSignal     :=0; (* 0: Signal=Low, 1: Signal=High, 2: always  *)
ST02_S1_70K61_A1.sInit.MaxTime         		:=2000;

(*ST02_S1_40K01 Freigabe Förderband von SPM (DigIn)*)
ST02_S1_40K01.sInit.InstName                :='ST02_S1_40K01';
ST02_S1_40K01.sInit.Description             :=' Freigabe Förderband von SPM';
ST02_S1_40K01.sInit.BitInName               :='-S1_40K01_14';
ST02_S1_40K01.sInit.HomePosSignal    :=2; (* 0: Signal=Low, 1: Signal=High, 2: always  *)
ST02_S1_40K01.sInit.MaxTime                 :=2000;

(* Init ST02_FDB_80_B02 Band Entnahmeposition 2  (DigIn) *)
ST02_FDB_80_B02.sInit.InstName                :='ST02_FDB_80_B02';
ST02_FDB_80_B02.sInit.Description             :=' Band Entnahmeposition 2';
ST02_FDB_80_B02.sInit.BitInName               :='-80_B02';
ST02_FDB_80_B02.sInit.HomePosSignal    :=2; (* 0: Signal=Low, 1: Signal=High, 2: always  *)
ST02_FDB_80_B02.sInit.MaxTime                 :=2000;

(* Init ST02_35_S31 ST02 Druckschalter Wartungseinheit Hauptluft min.6 bar (DigIn) *)
ST02_35_S31.sInit.InstName            :='ST02_35_S31';
ST02_35_S31.sInit.Description         :='ST02 Druckschalter Wartungseinheit Hauptluft min.6 bar';
ST02_35_S31.sInit.BitInName           :='-35_S31';
ST02_35_S31.sInit.HomePosSignal       :=2; (* 0: Signal=Low, 1: Signal=High, 2: always  *)
ST02_35_S31.sInit.MaxTime             :=2000;
ST02_35_S31.sInit.EnableInEveryMode   :=TRUE;

(*---------------------------------------------------------------------------------------------------------------*)
(* Init ST02_62_Y6 Tisch drehen 0 - 180 Grad(Valve) *)
ST02_62_Y6.sInit.InstName            :='ST02_62_Y6';
ST02_62_Y6.sInit.BitName            :='+62Y6';
ST02_62_Y6.sInit.Description         :='Tisch drehen ';
ST02_62_Y6.sInit.HomePosDefine       :=HOME_ALWAYS;
ST02_62_Y6.sInit.InitDescription     :='0 Grad';
ST02_62_Y6.sInit.WorkDescription     :='180 Grad';
ST02_62_Y6.sInit.DampBothTime        :=200;
ST02_62_Y6.sInit.KindOfValve         :='2G';
ST02_62_Y6.sInit.MaxTime             :=2000;

(* Init ST02_FDB_40_B61 Iso von SPM auf Band abgelegt (DigIn) *)
ST02_FDB_40_B61.sInit.InstName            :='ST02_FDB_40_B61';
ST02_FDB_40_B61.sInit.Description         :=' Iso von SPM auf Band abgelegt';
ST02_FDB_40_B61.sInit.BitInName           :='+40B61';
ST02_FDB_40_B61.sInit.HomePosSignal       :=2; (* 0: Signal=Low, 1: Signal=High, 2: always  *)
ST02_FDB_40_B61.sInit.MaxTime             :=2000;
(*ST02_FDB_40_B61.sInit.EnableInEveryMode   :=FALSE;*)

(* Init ST02_FDB_40_B71 Iso auf Band vor Vereinzler (DigIn) *)
ST02_FDB_40_B71.sInit.InstName            :='ST02_FDB_40_B71';
ST02_FDB_40_B71.sInit.Description         :=' Iso auf Band vor Vereinzler';
ST02_FDB_40_B71.sInit.BitInName           :='+40B71';
ST02_FDB_40_B71.sInit.HomePosSignal       :=2; (* 0: Signal=Low, 1: Signal=High, 2: always  *)
ST02_FDB_40_B71.sInit.MaxTime             :=2000;
(*ST02_FDB_40_B71.sInit.EnableInEveryMode   :=FALSE;*)

(* Init ST02_DT_62_B81 Tisch drehen 0 Grad (ValveSensor) *)
ST02_DT_62_B81.sInit.InstName            :='ST02_DT_62_B81';
ST02_DT_62_B81.sInit.BitName            :='+62B81';
ST02_DT_62_B81.sInit.Description         :='Tisch drehen 0 Grad';
ST02_DT_62_B81.sInit.SensorType          :=sValveSensorType_INIT;

(* Init ST02_DT_62_B91 Tisch drehen 180 Grad (ValveSensor) *)
ST02_DT_62_B91.sInit.InstName            :='ST02_DT_62_B91';
ST02_DT_62_B91.sInit.BitName            :='+62B91';
ST02_DT_62_B91.sInit.Description         :='Tisch drehen 180 Grad';
ST02_DT_62_B91.sInit.SensorType          :=sValveSensorType_WORK;

(*---------------------------------------------------------------------------------------------------------------*)
(* Init ST02_62_Y9 Schwenkarm 2 drehen 90 - 180 Grad(Valve) *)
ST02_62_Y9.sInit.InstName            :='ST02_62_Y9';
ST02_62_Y9.sInit.BitName            :='+62Y9';
ST02_62_Y9.sInit.Description         :='Schwenkarm 2 drehen 90 - 180 Grad ';
ST02_62_Y9.sInit.HomePosDefine       :=HOME_ALWAYS;
ST02_62_Y9.sInit.InitDescription     :='90 Grad';
ST02_62_Y9.sInit.WorkDescription     :='180 Grad';
ST02_62_Y9.sInit.DampBothTime        :=200;
ST02_62_Y9.sInit.KindOfValve         :='2G';
ST02_62_Y9.sInit.MaxTime             :=2000;

(* Init ST02_62_Y11 Schwenkarm 2 drehen 90 - 0 Grad(Valve) *)
ST02_62_Y11.sInit.InstName            :='ST02_62_Y11';
ST02_62_Y11.sInit.BitName            :='+62Y11';
ST02_62_Y11.sInit.Description         :='Schwenkarm 2 drehen 90 - 0 Grad ';
ST02_62_Y11.sInit.HomePosDefine       :=HOME_ALWAYS;
ST02_62_Y11.sInit.InitDescription     :='90 Grad';
ST02_62_Y11.sInit.WorkDescription     :='0 Grad';
ST02_62_Y11.sInit.DampBothTime        :=200;
ST02_62_Y11.sInit.KindOfValve         :='2G';
ST02_62_Y11.sInit.MaxTime             :=2000;

(* Init ST02_DT_61_B31 Schwenkarm 2 0 Grad (ValveSensor) *)
ST02_DT_61_B31.sInit.InstName            :='ST02_DT_61_B31';
ST02_DT_61_B31.sInit.BitName            :='+61B31';
ST02_DT_61_B31.sInit.Description         :='Schwenkarm 2 0 Grad';
ST02_DT_61_B31.sInit.SensorType          :=sValveSensorType_WORK;

(* Init ST02_DT_61_B11 Schwenkarm 2 180 Grad (ValveSensor) *)
ST02_DT_61_B11.sInit.InstName            :='ST02_DT_61_B11';
ST02_DT_61_B11.sInit.BitName            :='+61B11';
ST02_DT_61_B11.sInit.Description         :='Schwenkarm 2 180 Grad';
ST02_DT_61_B11.sInit.SensorType          :=sValveSensorType_WORK;

(*---------------------------------------------------------------------------------------------------------------*)
(* Init ST02_62_Y13 Schwenkarm 1 drehen 90 - 180 Grad(Valve) *)
ST02_62_Y13.sInit.InstName            :='ST02_62_Y13';
ST02_62_Y13.sInit.BitName            :='+62Y13';
ST02_62_Y13.sInit.Description         :='Schwenkarm 1 drehen 90 - 180 Grad ';
ST02_62_Y13.sInit.HomePosDefine       :=HOME_ALWAYS;
ST02_62_Y13.sInit.InitDescription     :='90 Grad';
ST02_62_Y13.sInit.WorkDescription     :='180 Grad';
ST02_62_Y13.sInit.DampBothTime        :=200;
ST02_62_Y13.sInit.KindOfValve         :='2G';
ST02_62_Y13.sInit.MaxTime             :=2000;

(* Init ST02_62_Y15 Schwenkarm 1 drehen 90 - 0 Grad(Valve) *)
ST02_62_Y15.sInit.InstName            :='ST02_62_Y15';
ST02_62_Y15.sInit.BitName            :='+62Y15';
ST02_62_Y15.sInit.Description         :='Schwenkarm 1 drehen 90 - 0 Grad ';
ST02_62_Y15.sInit.HomePosDefine       :=HOME_ALWAYS;
ST02_62_Y15.sInit.InitDescription     :='90 Grad';
ST02_62_Y15.sInit.WorkDescription     :='0 Grad';
ST02_62_Y15.sInit.DampBothTime        :=200;
ST02_62_Y15.sInit.KindOfValve         :='2G';
ST02_62_Y15.sInit.MaxTime             :=2000;

(* Init ST02_DT_62_B11 Schwenkarm 1 0 Grad (ValveSensor) *)
ST02_DT_62_B11.sInit.InstName            :='ST02_DT_62_B11';
ST02_DT_62_B11.sInit.BitName            :='+62B11';
ST02_DT_62_B11.sInit.Description         :='Schwenkarm 1 0 Grad';
ST02_DT_62_B11.sInit.SensorType          :=sValveSensorType_WORK;

(* Init ST02_DT_61_B41 Schwenkarm 1 180 Grad (ValveSensor) *)
ST02_DT_61_B41.sInit.InstName            :='ST02_DT_61_B41';
ST02_DT_61_B41.sInit.BitName            :='+61B41';
ST02_DT_61_B41.sInit.Description         :='Schwenkarm 2 180 Grad';
ST02_DT_61_B41.sInit.SensorType          :=sValveSensorType_WORK;

(* Init ST02_62_Y4 Kamera Ausschleusen Bandstrecke (Valve) *)
ST02_62_Y4.sInit.InstName            :='ST02_62_Y4';
ST02_62_Y4.sInit.BitName            :='+62Y4';
ST02_62_Y4.sInit.Description         :='Kamera Ausschleusen';
ST02_62_Y4.sInit.HomePosDefine       :=HOME_ALWAYS;
ST02_62_Y4.sInit.InitDescription     :='GS';
ST02_62_Y4.sInit.WorkDescription     :='AS';
ST02_62_Y4.sInit.DampBothTime        :=200;
ST02_62_Y4.sInit.KindOfValve         :='2G';
ST02_62_Y4.sInit.MaxTime             :=4000;

(* Init ST02_FDB_54_B11 Kamera Ausschleusen Bandstrecke eingefahren (ValveSensor) *)
ST02_FDB_54_B11.sInit.InstName            :='ST02_FDB_54_B11';
ST02_FDB_54_B11.sInit.BitName            :='+54B11';
ST02_FDB_54_B11.sInit.Description         :='Kamera Ausschleusen';
ST02_FDB_54_B11.sInit.SensorType          :=sValveSensorType_INIT;

(* Init ST02_FDB_54_B21 Kamera Ausschleusen Bandstrecke ausgefahren (ValveSensor) *)
ST02_FDB_54_B21.sInit.InstName            :='ST02_FDB_54_B21';
ST02_FDB_54_B21.sInit.BitName            :='+54B21';
ST02_FDB_54_B21.sInit.Description         :='Kamera Ausschleusen';
ST02_FDB_54_B21.sInit.SensorType          :=sValveSensorType_WORK;



(*Init ST02_62_Y17 Schwenkarm 1 ISK Fixierung ein/ausfahren(Valve) *)
ST02_62_Y17.sInit.InstName            :='ST02_62_Y17';
ST02_62_Y17.sInit.BitName            :='+62_Y17';
ST02_62_Y17.sInit.Description         :='Iso 1 fiexieren';
ST02_62_Y17.sInit.HomePosDefine       :=HOME_ALWAYS;
ST02_62_Y17.sInit.InitDescription     :='GS';
ST02_62_Y17.sInit.WorkDescription     :='AS';
ST02_62_Y17.sInit.DampBothTime        :=200;
ST02_62_Y17.sInit.KindOfValve         :='2G';
ST02_62_Y17.sInit.MaxTime             :=4000;

(* Init ST02_S1_66_B11 Schwenkarm 1 ISK Fixierung GST (ValveSensor) *)
ST02_S1_66_B11.sInit.InstName            :='ST02_S1_66_B21';
ST02_S1_66_B11.sInit.BitName            :='+S1_66B11';
ST02_S1_66_B11.sInit.Description         :='Iso fixieren';
ST02_S1_66_B11.sInit.SensorType          :=sValveSensorType_INIT;

(* Init ST02_S1_66_B21 Schwenkarm 1 ISK Fixierung AST (ValveSensor) *)
ST02_S1_66_B21.sInit.InstName            :='ST02_S1_66_B21';
ST02_S1_66_B21.sInit.BitName            :='+S1_66B21';
ST02_S1_66_B21.sInit.Description         :='Iso fixieren';
ST02_S1_66_B21.sInit.SensorType          :=sValveSensorType_WORK;


(*Init ST02_62_Y18 Schwenkarm 2 ISK Fixierung ein/ausfahren(Valve) (Valve) *)
ST02_62_Y18.sInit.InstName            :='ST02_62_Y18';
ST02_62_Y18.sInit.BitName            :='+62_Y18';
ST02_62_Y18.sInit.Description         :='Iso 2 fiexieren';
ST02_62_Y18.sInit.HomePosDefine       :=HOME_ALWAYS;
ST02_62_Y18.sInit.InitDescription     :='GS';
ST02_62_Y18.sInit.WorkDescription     :='AS';
ST02_62_Y18.sInit.DampBothTime        :=200;
ST02_62_Y18.sInit.KindOfValve         :='2G';
ST02_62_Y18.sInit.MaxTime             :=4000;

(* Init ST02_S1_66_B31 Schwenkarm 2 ISK Fixierung GST (ValveSensor) *)
ST02_S1_66_B31.sInit.InstName            :='ST02_S1_66_B31';
ST02_S1_66_B31.sInit.BitName            :='S1_66B31';
ST02_S1_66_B31.sInit.Description         :='Iso fixieren';
ST02_S1_66_B31.sInit.SensorType          :=sValveSensorType_INIT;

(* Init ST02_S1_66_B41 Schwenkarm 2 ISK Fixierung AST (ValveSensor) *)
ST02_S1_66_B41.sInit.InstName            :='ST02_S1_66_B41';
ST02_S1_66_B41.sInit.BitName            :='S1_66_B41';
ST02_S1_66_B41.sInit.Description         :='Iso fixieren';
ST02_S1_66_B41.sInit.SensorType          :=sValveSensorType_WORK;


(* Init ST02_35Y01 Einschaltventil Hauptluft Tampondruckanlage (Valve) *)
ST02_35Y01.sInit.InstName          :='ST02_35Y01';
ST02_35Y01.sInit.BitName          :='+35Y01';
ST02_35Y01.sInit.Description       :='Hauptluft Tampondrucker';
ST02_35Y01.sInit.HomePosDefine     :=HOME_ALWAYS;
ST02_35Y01.sInit.InitDescription   :='GS';
ST02_35Y01.sInit.WorkDescription   :='AS';
ST02_35Y01.sInit.DampBothTime      :=0;
ST02_35Y01.sInit.MaxTime           :=2000;
ST02_35Y01.sInit.KindOfValve       :='A';
END_PROGRAM

(* POU Stations/ST_03_Ruestsaetze/ST_03__Init/ST03_Init, ST *)
PROGRAM ST03_Init


VAR


	sDigInVisu: BOOL;
END_VAR
(*INIT Aufrufe für Rüstsätze*)
Init_154polRP();	Init_154pol();
Init_160pol();		Init_206pol();
Init_92pol();		Init_124pol();
Init_46pol();		Init_NOX5_6pol();
Init_NOX4pol();	Init_88pol();
Init_7pol();		Init_88polAMG();
Init_120pol();		Init_21pol();
Init_191pol();		Init_48pol();
Init_72pol();		Init_268pol_102pol_neu();
Init_268polRP();	Init_33pol();

(* ----------------------------------------------------------------------------------------- *)
IF NOT MP.ST03.SGM_3621 THEN
	(*Init ST03_51_M1 Förderbandmotor*)
	ST03_51_M1.sConfig.Description		:='Förderband';
	ST03_51_M1.sConfig.InstName			:='ST03_51_M1';
	ST03_51_M1.sConfig.Aktiv				:=TRUE;
	ST03_51_M1.sConfig.Skalierfaktor		:=360.0 / (EXPT(2,20))	; (*360°/ 20 bit Encoder =0.00034332275390625*)
	ST03_51_M1.sConfig.Getriebefaktor		:=25;
	ST03_51_M1.sConfig.Modulo			:=FALSE;
	ST03_51_M1.sConfig.Pos_Faktor		:=157.07;			(*Weg bei einer Umdrehung in mm (nach Getriebe)*)
	ST03_51_M1.sConfig.maxRpm			:=5338;
	ST03_51_M1.sConfig.ModeOfOperation	:=CSP;				(*CSP,CSV,CST,CSTCA muss an der KLemme (Coe-Online 7010.03) eingestellt werden*)
	(*(CSP) position mode*)
	ST03_51_M1.sConfig.Torque_Limit		:=0;			(*bei 0 ausgeschaltet*)
	ST03_51_M1.sConfig.SW_Limit_on		:=FALSE;
	ST03_51_M1.sConfig.SW_Limit_min		:=-EXPT(2,32);
	ST03_51_M1.sConfig.SW_Limit_max		:=EXPT(2,32);
	ST03_51_M1.sConfig.lr_kp 				:= 800;
	ST03_51_M1.sConfig.lr_ki 				:= 100.0;
	ST03_51_M1.sConfig.lr_kd 				:= 50;
ELSE
	(* Init ST03_A5 Bandantrieb Förderbandmotor Oriental (nur 3621) Ein (DigOutIn)   ST08_170_K2 *)
	ST03_A5.sInit.InstName               :='ST03_A5';
	ST03_A5.sInit.Description            :='Förderbandmotor Isokörper';
	ST03_A5.sInit.BitOutName             :='-3_A5';
	ST03_A5.sInit.BitInName              :='';
	ST03_A5.sInit.HomePosOutput          :=2; (* 0: Signal=Low, 1: Signal=High, 2: always  *)
	ST03_A5.sInit.MaxTime                :=2000;
	ST03_A5.sInit.EnableInEveryMode  :=TRUE;
END_IF

(* Init ST03_V2 Störung Motor Förderband Oriental (DigIn) *)
ST03_V2.sInit.InstName               :='ST03_V2';
ST03_V2.sInit.Description            :='Störung Motor Förderband';
ST03_V2.sInit.BitInName              :='+3-V2';
ST03_V2.sInit.HomePosSignal          :=2; (* 0: Signal=Low, 1: Signal=High, 2: always  *)
ST03_V2.sInit.MaxTime                :=10;
ST03_V2.sInit.EnableInEveryMode       :=TRUE;

(* Init ST03_601V1_A1  Förderband Prüfteile (DigOutIn)  *)
ST03_601V1_A1.sInit.InstName               :='ST03_601V1_A1';
ST03_601V1_A1.sInit.Description            :='Förderband Prüfteile';
ST03_601V1_A1.sInit.BitOutName             :='-60V1_A1';
ST03_601V1_A1.sInit.BitInName              :='';
ST03_601V1_A1.sInit.HomePosOutput          :=2; (* 0: Signal=Low, 1: Signal=High, 2: always  *)
ST03_601V1_A1.sInit.MaxTime                :=2000;
ST03_601V1_A1.sInit.EnableInEveryMode  			:=TRUE;

(* ----------------------------------------------------------------------------------------- *)
(* 																	Roboter																									 *)
(* ----------------------------------------------------------------------------------------- *)
Visu.Robot01.TcpIpAdress:=MP.ST03.RobotIPAdress;
Robot01.sInit.InstName				:='Robot01';
Robot01.sInit.BitName				:='+3-125_A1';
Robot01.sInit.Description				:='ST03 Roboter';
Robot01.sInit.TcpIPAdress			:=MP.ST03.RobotIPAdress; (*10.16.55.130*)
Robot01.sInit.TcpIPSocket			:=2000;
Robot01.sInit.MaxTime				:=40000;
Robot01.sInit.WithToolHandling		:=TRUE;
Robot01.sInit.ToolMaxTime			:=2000;

